LIN {X 108.19, Y 113.72, Z 0.00, A 0, B 0, C 0} C_DIS
LIN {X 108.38, Y 113.55, Z 0.00, A 0, B 0, C 0} C_DIS
LIN {X 108.56, Y 113.38, Z 0.00, A 0, B 0, C 0} C_DIS
LIN {X 108.74, Y 113.19, Z 0.00, A 0, B 0, C 0} C_DIS
LIN {X 108.92, Y 113.00, Z 0.00, A 0, B 0, C 0} C_DIS
LIN {X 109.10, Y 112.81, Z 0.00, A 0, B 0, C 0} C_DIS
LIN {X 109.28, Y 112.63, Z 0.00, A 0, B 0, C 0} C_DIS
LIN {X 109.46, Y 112.45, Z 0.00, A 0, B 0, C 0} C_DIS
LIN {X 109.65, Y 112.29, Z 0.00, A 0, B 0, C 0} C_DIS
LIN {X 109.84, Y 112.14, Z 0.00, A 0, B 0, C 0} C_DIS
LIN {X 110.04, Y 112.00, Z 0.00, A 0, B 0, C 0} C_DIS
LIN {X 110.23, Y 111.86, Z 0.00, A 0, B 0, C 0} C_DIS
LIN {X 110.42, Y 111.71, Z 0.00, A 0, B 0, C 0} C_DIS
LIN {X 110.61, Y 111.54, Z 0.00, A 0, B 0, C 0} C_DIS
LIN {X 110.79, Y 111.36, Z 0.00, A 0, B 0, C 0} C_DIS
LIN {X 110.97, Y 111.17, Z 0.00, A 0, B 0, C 0} C_DIS
LIN {X 111.15, Y 110.98, Z 0.00, A 0, B 0, C 0} C_DIS
LIN {X 111.33, Y 110.79, Z 0.00, A 0, B 0, C 0} C_DIS
LIN {X 111.51, Y 110.61, Z 0.00, A 0, B 0, C 0} C_DIS
LIN {X 111.69, Y 110.43, Z 0.00, A 0, B 0, C 0} C_DIS
LIN {X 111.88, Y 110.27, Z 0.00, A 0, B 0, C 0} C_DIS
LIN {X 112.07, Y 110.13, Z 0.00, A 0, B 0, C 0} C_DIS
LIN {X 112.27, Y 110.00, Z 0.00, A 0, B 0, C 0} C_DIS
LIN {X 112.47, Y 109.86, Z 0.00, A 0, B 0, C 0} C_DIS
LIN {X 112.65, Y 109.69, Z 0.00, A 0, B 0, C 0} C_DIS
LIN {X 112.85, Y 109.53, Z 0.00, A 0, B 0, C 0} C_DIS
LIN {X 113.05, Y 109.41, Z 0.00, A 0, B 0, C 0} C_DIS
LIN {X 113.25, Y 109.28, Z 0.00, A 0, B 0, C 0} C_DIS
LIN {X 113.42, Y 109.10, Z 0.00, A 0, B 0, C 0} C_DIS
LIN {X 113.58, Y 108.88, Z 0.00, A 0, B 0, C 0} C_DIS
LIN {X 113.74, Y 108.65, Z 0.00, A 0, B 0, C 0} C_DIS
LIN {X 113.89, Y 108.41, Z 0.00, A 0, B 0, C 0} C_DIS
LIN {X 114.02, Y 108.15, Z 0.00, A 0, B 0, C 0} C_DIS
LIN {X 114.12, Y 107.87, Z 0.00, A 0, B 0, C 0} C_DIS
LIN {X 114.20, Y 107.57, Z 0.00, A 0, B 0, C 0} C_DIS
LIN {X 114.26, Y 107.25, Z 0.00, A 0, B 0, C 0} C_DIS
LIN {X 114.30, Y 106.92, Z 0.00, A 0, B 0, C 0} C_DIS
LIN {X 114.33, Y 106.60, Z 0.00, A 0, B 0, C 0} C_DIS
LIN {X 114.36, Y 106.27, Z 0.00, A 0, B 0, C 0} C_DIS
LIN {X 114.38, Y 105.95, Z 0.00, A 0, B 0, C 0} C_DIS
LIN {X 114.39, Y 105.62, Z 0.00, A 0, B 0, C 0} C_DIS
LIN {X 114.39, Y 105.30, Z 0.00, A 0, B 0, C 0} C_DIS
LIN {X 114.40, Y 104.97, Z 0.00, A 0, B 0, C 0} C_DIS
LIN {X 114.39, Y 104.64, Z 0.00, A 0, B 0, C 0} C_DIS
LIN {X 114.39, Y 104.31, Z 0.00, A 0, B 0, C 0} C_DIS
LIN {X 114.39, Y 103.99, Z 0.00, A 0, B 0, C 0} C_DIS
LIN {X 114.38, Y 103.66, Z 0.00, A 0, B 0, C 0} C_DIS
LIN {X 114.38, Y 103.33, Z 0.00, A 0, B 0, C 0} C_DIS
LIN {X 114.38, Y 103.00, Z 0.00, A 0, B 0, C 0} C_DIS
LIN {X 114.38, Y 102.67, Z 0.00, A 0, B 0, C 0} C_DIS
LIN {X 114.38, Y 102.35, Z 0.00, A 0, B 0, C 0} C_DIS
LIN {X 114.38, Y 102.02, Z 0.00, A 0, B 0, C 0} C_DIS
LIN {X 114.39, Y 101.69, Z 0.00, A 0, B 0, C 0} C_DIS
LIN {X 114.39, Y 101.36, Z 0.00, A 0, B 0, C 0} C_DIS
LIN {X 114.39, Y 101.04, Z 0.00, A 0, B 0, C 0} C_DIS
LIN {X 114.39, Y 100.71, Z 0.00, A 0, B 0, C 0} C_DIS
LIN {X 114.39, Y 100.38, Z 0.00, A 0, B 0, C 0} C_DIS
LIN {X 114.39, Y 100.05, Z 0.00, A 0, B 0, C 0} C_DIS
LIN {X 114.39, Y 99.73, Z 0.00, A 0, B 0, C 0} C_DIS
LIN {X 114.38, Y 99.40, Z 0.00, A 0, B 0, C 0} C_DIS
LIN {X 114.38, Y 99.07, Z 0.00, A 0, B 0, C 0} C_DIS
LIN {X 114.38, Y 98.74, Z 0.00, A 0, B 0, C 0} C_DIS
LIN {X 114.38, Y 98.41, Z 0.00, A 0, B 0, C 0} C_DIS
LIN {X 114.38, Y 98.08, Z 0.00, A 0, B 0, C 0} C_DIS
LIN {X 114.39, Y 97.76, Z 0.00, A 0, B 0, C 0} C_DIS
LIN {X 114.40, Y 97.43, Z 0.00, A 0, B 0, C 0} C_DIS
LIN {X 114.42, Y 97.11, Z 0.00, A 0, B 0, C 0} C_DIS
LIN {X 114.46, Y 96.79, Z 0.00, A 0, B 0, C 0} C_DIS
LIN {X 114.54, Y 96.49, Z 0.00, A 0, B 0, C 0} C_DIS
LIN {X 114.67, Y 96.21, Z 0.00, A 0, B 0, C 0} C_DIS
LIN {X 114.82, Y 95.97, Z 0.00, A 0, B 0, C 0} C_DIS
LIN {X 115.00, Y 95.78, Z 0.00, A 0, B 0, C 0} C_DIS
LIN {X 115.19, Y 95.65, Z 0.00, A 0, B 0, C 0} C_DIS
LIN {X 115.40, Y 95.57, Z 0.00, A 0, B 0, C 0} C_DIS
LIN {X 115.61, Y 95.48, Z 0.00, A 0, B 0, C 0} C_DIS
LIN {X 115.81, Y 95.35, Z 0.00, A 0, B 0, C 0} C_DIS
LIN {X 116.01, Y 95.22, Z 0.00, A 0, B 0, C 0} C_DIS
LIN {X 116.22, Y 95.12, Z 0.00, A 0, B 0, C 0} C_DIS
LIN {X 116.43, Y 95.03, Z 0.00, A 0, B 0, C 0} C_DIS
LIN {X 116.63, Y 94.92, Z 0.00, A 0, B 0, C 0} C_DIS
LIN {X 116.83, Y 94.78, Z 0.00, A 0, B 0, C 0} C_DIS
LIN {X 117.01, Y 94.61, Z 0.00, A 0, B 0, C 0} C_DIS
LIN {X 117.20, Y 94.45, Z 0.00, A 0, B 0, C 0} C_DIS
LIN {X 117.40, Y 94.32, Z 0.00, A 0, B 0, C 0} C_DIS
LIN {X 117.60, Y 94.20, Z 0.00, A 0, B 0, C 0} C_DIS
LIN {X 117.79, Y 94.04, Z 0.00, A 0, B 0, C 0} C_DIS
LIN {X 117.97, Y 93.86, Z 0.00, A 0, B 0, C 0} C_DIS
LIN {X 118.15, Y 93.67, Z 0.00, A 0, B 0, C 0} C_DIS
LIN {X 118.33, Y 93.49, Z 0.00, A 0, B 0, C 0} C_DIS
LIN {X 118.52, Y 93.31, Z 0.00, A 0, B 0, C 0} C_DIS
LIN {X 118.70, Y 93.13, Z 0.00, A 0, B 0, C 0} C_DIS
LIN {X 118.88, Y 92.95, Z 0.00, A 0, B 0, C 0} C_DIS
LIN {X 119.06, Y 92.77, Z 0.00, A 0, B 0, C 0} C_DIS
LIN {X 119.24, Y 92.59, Z 0.00, A 0, B 0, C 0} C_DIS
LIN {X 119.42, Y 92.40, Z 0.00, A 0, B 0, C 0} C_DIS
LIN {X 119.60, Y 92.22, Z 0.00, A 0, B 0, C 0} C_DIS
LIN {X 119.78, Y 92.03, Z 0.00, A 0, B 0, C 0} C_DIS
LIN {X 119.96, Y 91.85, Z 0.00, A 0, B 0, C 0} C_DIS
LIN {X 120.14, Y 91.67, Z 0.00, A 0, B 0, C 0} C_DIS
LIN {X 120.33, Y 91.50, Z 0.00, A 0, B 0, C 0} C_DIS
LIN {X 120.51, Y 91.32, Z 0.00, A 0, B 0, C 0} C_DIS
LIN {X 120.70, Y 91.14, Z 0.00, A 0, B 0, C 0} C_DIS
LIN {X 120.87, Y 90.96, Z 0.00, A 0, B 0, C 0} C_DIS
LIN {X 121.04, Y 90.76, Z 0.00, A 0, B 0, C 0} C_DIS
LIN {X 121.21, Y 90.54, Z 0.00, A 0, B 0, C 0} C_DIS
LIN {X 121.36, Y 90.32, Z 0.00, A 0, B 0, C 0} C_DIS
LIN {X 121.52, Y 90.08, Z 0.00, A 0, B 0, C 0} C_DIS
LIN {X 121.67, Y 89.85, Z 0.00, A 0, B 0, C 0} C_DIS
LIN {X 121.83, Y 89.63, Z 0.00, A 0, B 0, C 0} C_DIS
LIN {X 121.99, Y 89.41, Z 0.00, A 0, B 0, C 0} C_DIS
LIN {X 122.16, Y 89.21, Z 0.00, A 0, B 0, C 0} C_DIS
LIN {X 122.34, Y 89.02, Z 0.00, A 0, B 0, C 0} C_DIS
LIN {X 122.52, Y 88.84, Z 0.00, A 0, B 0, C 0} C_DIS
LIN {X 122.71, Y 88.67, Z 0.00, A 0, B 0, C 0} C_DIS
LIN {X 122.89, Y 88.49, Z 0.00, A 0, B 0, C 0} C_DIS
LIN {X 123.07, Y 88.31, Z 0.00, A 0, B 0, C 0} C_DIS
LIN {X 123.24, Y 88.11, Z 0.00, A 0, B 0, C 0} C_DIS
LIN {X 123.41, Y 87.90, Z 0.00, A 0, B 0, C 0} C_DIS
LIN {X 123.56, Y 87.67, Z 0.00, A 0, B 0, C 0} C_DIS
LIN {X 123.72, Y 87.44, Z 0.00, A 0, B 0, C 0} C_DIS
LIN {X 123.87, Y 87.20, Z 0.00, A 0, B 0, C 0} C_DIS
LIN {X 124.01, Y 86.95, Z 0.00, A 0, B 0, C 0} C_DIS
LIN {X 124.13, Y 86.68, Z 0.00, A 0, B 0, C 0} C_DIS
LIN {X 124.24, Y 86.40, Z 0.00, A 0, B 0, C 0} C_DIS
LIN {X 124.36, Y 86.13, Z 0.00, A 0, B 0, C 0} C_DIS
LIN {X 124.48, Y 85.85, Z 0.00, A 0, B 0, C 0} C_DIS
LIN {X 124.60, Y 85.58, Z 0.00, A 0, B 0, C 0} C_DIS
LIN {X 124.73, Y 85.32, Z 0.00, A 0, B 0, C 0} C_DIS
LIN {X 124.87, Y 85.06, Z 0.00, A 0, B 0, C 0} C_DIS
LIN {X 125.01, Y 84.82, Z 0.00, A 0, B 0, C 0} C_DIS
LIN {X 125.16, Y 84.58, Z 0.00, A 0, B 0, C 0} C_DIS
LIN {X 125.31, Y 84.35, Z 0.00, A 0, B 0, C 0} C_DIS
LIN {X 125.47, Y 84.12, Z 0.00, A 0, B 0, C 0} C_DIS
LIN {X 125.63, Y 83.90, Z 0.00, A 0, B 0, C 0} C_DIS
LIN {X 125.79, Y 83.67, Z 0.00, A 0, B 0, C 0} C_DIS
LIN {X 125.94, Y 83.44, Z 0.00, A 0, B 0, C 0} C_DIS
LIN {X 126.08, Y 83.19, Z 0.00, A 0, B 0, C 0} C_DIS
LIN {X 126.22, Y 82.93, Z 0.00, A 0, B 0, C 0} C_DIS
LIN {X 126.34, Y 82.67, Z 0.00, A 0, B 0, C 0} C_DIS
LIN {X 126.46, Y 82.39, Z 0.00, A 0, B 0, C 0} C_DIS
LIN {X 126.57, Y 82.11, Z 0.00, A 0, B 0, C 0} C_DIS
LIN {X 126.68, Y 81.83, Z 0.00, A 0, B 0, C 0} C_DIS
LIN {X 126.77, Y 81.53, Z 0.00, A 0, B 0, C 0} C_DIS
LIN {X 126.85, Y 81.23, Z 0.00, A 0, B 0, C 0} C_DIS
LIN {X 126.95, Y 80.94, Z 0.00, A 0, B 0, C 0} C_DIS
LIN {X 127.07, Y 80.66, Z 0.00, A 0, B 0, C 0} C_DIS
LIN {X 127.19, Y 80.39, Z 0.00, A 0, B 0, C 0} C_DIS
LIN {X 127.31, Y 80.12, Z 0.00, A 0, B 0, C 0} C_DIS
LIN {X 127.43, Y 79.85, Z 0.00, A 0, B 0, C 0} C_DIS
LIN {X 127.56, Y 79.58, Z 0.00, A 0, B 0, C 0} C_DIS
LIN {X 127.68, Y 79.31, Z 0.00, A 0, B 0, C 0} C_DIS
LIN {X 127.80, Y 79.03, Z 0.00, A 0, B 0, C 0} C_DIS
LIN {X 127.91, Y 78.75, Z 0.00, A 0, B 0, C 0} C_DIS
LIN {X 128.01, Y 78.46, Z 0.00, A 0, B 0, C 0} C_DIS
LIN {X 128.10, Y 78.16, Z 0.00, A 0, B 0, C 0} C_DIS
LIN {X 128.18, Y 77.86, Z 0.00, A 0, B 0, C 0} C_DIS
LIN {X 128.29, Y 77.58, Z 0.00, A 0, B 0, C 0} C_DIS
LIN {X 128.40, Y 77.30, Z 0.00, A 0, B 0, C 0} C_DIS
LIN {X 128.49, Y 77.00, Z 0.00, A 0, B 0, C 0} C_DIS
LIN {X 128.55, Y 76.69, Z 0.00, A 0, B 0, C 0} C_DIS
LIN {X 128.61, Y 76.37, Z 0.00, A 0, B 0, C 0} C_DIS
LIN {X 128.69, Y 76.06, Z 0.00, A 0, B 0, C 0} C_DIS
LIN {X 128.78, Y 75.77, Z 0.00, A 0, B 0, C 0} C_DIS
LIN {X 128.86, Y 75.46, Z 0.00, A 0, B 0, C 0} C_DIS
LIN {X 128.91, Y 75.14, Z 0.00, A 0, B 0, C 0} C_DIS
LIN {X 128.97, Y 74.83, Z 0.00, A 0, B 0, C 0} C_DIS
LIN {X 129.07, Y 74.54, Z 0.00, A 0, B 0, C 0} C_DIS
LIN {X 129.19, Y 74.26, Z 0.00, A 0, B 0, C 0} C_DIS
LIN {X 129.29, Y 73.97, Z 0.00, A 0, B 0, C 0} C_DIS
LIN {X 129.37, Y 73.67, Z 0.00, A 0, B 0, C 0} C_DIS
LIN {X 129.43, Y 73.36, Z 0.00, A 0, B 0, C 0} C_DIS
LIN {X 129.49, Y 73.04, Z 0.00, A 0, B 0, C 0} C_DIS
LIN {X 129.54, Y 72.72, Z 0.00, A 0, B 0, C 0} C_DIS
LIN {X 129.59, Y 72.40, Z 0.00, A 0, B 0, C 0} C_DIS
LIN {X 129.64, Y 72.08, Z 0.00, A 0, B 0, C 0} C_DIS
LIN {X 129.69, Y 71.76, Z 0.00, A 0, B 0, C 0} C_DIS
LIN {X 129.75, Y 71.45, Z 0.00, A 0, B 0, C 0} C_DIS
LIN {X 129.80, Y 71.13, Z 0.00, A 0, B 0, C 0} C_DIS
LIN {X 129.85, Y 70.81, Z 0.00, A 0, B 0, C 0} C_DIS
LIN {X 129.90, Y 70.49, Z 0.00, A 0, B 0, C 0} C_DIS
LIN {X 129.96, Y 70.18, Z 0.00, A 0, B 0, C 0} C_DIS
LIN {X 130.01, Y 69.86, Z 0.00, A 0, B 0, C 0} C_DIS
LIN {X 130.06, Y 69.54, Z 0.00, A 0, B 0, C 0} C_DIS
LIN {X 130.12, Y 69.22, Z 0.00, A 0, B 0, C 0} C_DIS
LIN {X 130.17, Y 68.90, Z 0.00, A 0, B 0, C 0} C_DIS
LIN {X 130.23, Y 68.59, Z 0.00, A 0, B 0, C 0} C_DIS
LIN {X 130.28, Y 68.27, Z 0.00, A 0, B 0, C 0} C_DIS
LIN {X 130.33, Y 67.95, Z 0.00, A 0, B 0, C 0} C_DIS
LIN {X 130.38, Y 67.63, Z 0.00, A 0, B 0, C 0} C_DIS
LIN {X 130.42, Y 67.31, Z 0.00, A 0, B 0, C 0} C_DIS
LIN {X 130.45, Y 66.99, Z 0.00, A 0, B 0, C 0} C_DIS
LIN {X 130.48, Y 66.66, Z 0.00, A 0, B 0, C 0} C_DIS
LIN {X 130.49, Y 66.34, Z 0.00, A 0, B 0, C 0} C_DIS
LIN {X 130.49, Y 66.01, Z 0.00, A 0, B 0, C 0} C_DIS
LIN {X 130.49, Y 65.68, Z 0.00, A 0, B 0, C 0} C_DIS
LIN {X 130.48, Y 65.35, Z 0.00, A 0, B 0, C 0} C_DIS
LIN {X 130.47, Y 65.02, Z 0.00, A 0, B 0, C 0} C_DIS
LIN {X 130.47, Y 64.69, Z 0.00, A 0, B 0, C 0} C_DIS
LIN {X 130.47, Y 64.37, Z 0.00, A 0, B 0, C 0} C_DIS
LIN {X 130.48, Y 64.04, Z 0.00, A 0, B 0, C 0} C_DIS
LIN {X 130.50, Y 63.72, Z 0.00, A 0, B 0, C 0} C_DIS
LIN {X 130.54, Y 63.39, Z 0.00, A 0, B 0, C 0} C_DIS
LIN {X 130.58, Y 63.07, Z 0.00, A 0, B 0, C 0} C_DIS
LIN {X 130.64, Y 62.76, Z 0.00, A 0, B 0, C 0} C_DIS
LIN {X 130.70, Y 62.44, Z 0.00, A 0, B 0, C 0} C_DIS
LIN {X 130.76, Y 62.12, Z 0.00, A 0, B 0, C 0} C_DIS
LIN {X 130.81, Y 61.80, Z 0.00, A 0, B 0, C 0} C_DIS
LIN {X 130.85, Y 61.48, Z 0.00, A 0, B 0, C 0} C_DIS
LIN {X 130.88, Y 61.16, Z 0.00, A 0, B 0, C 0} C_DIS
LIN {X 130.90, Y 60.84, Z 0.00, A 0, B 0, C 0} C_DIS
LIN {X 130.91, Y 60.51, Z 0.00, A 0, B 0, C 0} C_DIS
LIN {X 130.91, Y 60.18, Z 0.00, A 0, B 0, C 0} C_DIS
LIN {X 130.92, Y 59.85, Z 0.00, A 0, B 0, C 0} C_DIS
LIN {X 130.92, Y 59.53, Z 0.00, A 0, B 0, C 0} C_DIS
LIN {X 130.92, Y 59.20, Z 0.00, A 0, B 0, C 0} C_DIS
LIN {X 130.92, Y 58.87, Z 0.00, A 0, B 0, C 0} C_DIS
LIN {X 130.92, Y 58.54, Z 0.00, A 0, B 0, C 0} C_DIS
LIN {X 130.92, Y 58.22, Z 0.00, A 0, B 0, C 0} C_DIS
LIN {X 130.91, Y 57.89, Z 0.00, A 0, B 0, C 0} C_DIS
LIN {X 130.91, Y 57.56, Z 0.00, A 0, B 0, C 0} C_DIS
LIN {X 130.91, Y 57.23, Z 0.00, A 0, B 0, C 0} C_DIS
LIN {X 130.91, Y 56.90, Z 0.00, A 0, B 0, C 0} C_DIS
LIN {X 130.91, Y 56.58, Z 0.00, A 0, B 0, C 0} C_DIS
LIN {X 130.91, Y 56.25, Z 0.00, A 0, B 0, C 0} C_DIS
LIN {X 130.91, Y 55.92, Z 0.00, A 0, B 0, C 0} C_DIS
LIN {X 130.91, Y 55.59, Z 0.00, A 0, B 0, C 0} C_DIS
LIN {X 130.91, Y 55.27, Z 0.00, A 0, B 0, C 0} C_DIS
LIN {X 130.91, Y 54.94, Z 0.00, A 0, B 0, C 0} C_DIS
LIN {X 130.91, Y 54.61, Z 0.00, A 0, B 0, C 0} C_DIS
LIN {X 130.91, Y 54.28, Z 0.00, A 0, B 0, C 0} C_DIS
LIN {X 130.91, Y 53.96, Z 0.00, A 0, B 0, C 0} C_DIS
LIN {X 130.91, Y 53.63, Z 0.00, A 0, B 0, C 0} C_DIS
LIN {X 130.91, Y 53.30, Z 0.00, A 0, B 0, C 0} C_DIS
LIN {X 130.91, Y 52.97, Z 0.00, A 0, B 0, C 0} C_DIS
LIN {X 130.91, Y 52.64, Z 0.00, A 0, B 0, C 0} C_DIS
LIN {X 130.91, Y 52.32, Z 0.00, A 0, B 0, C 0} C_DIS
LIN {X 130.91, Y 51.99, Z 0.00, A 0, B 0, C 0} C_DIS
LIN {X 130.91, Y 51.66, Z 0.00, A 0, B 0, C 0} C_DIS
LIN {X 130.91, Y 51.33, Z 0.00, A 0, B 0, C 0} C_DIS
LIN {X 130.91, Y 51.01, Z 0.00, A 0, B 0, C 0} C_DIS
LIN {X 130.91, Y 50.68, Z 0.00, A 0, B 0, C 0} C_DIS
LIN {X 130.91, Y 50.35, Z 0.00, A 0, B 0, C 0} C_DIS
LIN {X 130.91, Y 50.02, Z 0.00, A 0, B 0, C 0} C_DIS
LIN {X 130.91, Y 49.69, Z 0.00, A 0, B 0, C 0} C_DIS
LIN {X 130.91, Y 49.37, Z 0.00, A 0, B 0, C 0} C_DIS
LIN {X 130.91, Y 49.04, Z 0.00, A 0, B 0, C 0} C_DIS
LIN {X 130.91, Y 48.71, Z 0.00, A 0, B 0, C 0} C_DIS
LIN {X 130.91, Y 48.38, Z 0.00, A 0, B 0, C 0} C_DIS
LIN {X 130.91, Y 48.06, Z 0.00, A 0, B 0, C 0} C_DIS
LIN {X 130.91, Y 47.73, Z 0.00, A 0, B 0, C 0} C_DIS
LIN {X 130.91, Y 47.40, Z 0.00, A 0, B 0, C 0} C_DIS
LIN {X 130.91, Y 47.07, Z 0.00, A 0, B 0, C 0} C_DIS
LIN {X 130.91, Y 46.75, Z 0.00, A 0, B 0, C 0} C_DIS
LIN {X 130.91, Y 46.42, Z 0.00, A 0, B 0, C 0} C_DIS
LIN {X 130.91, Y 46.09, Z 0.00, A 0, B 0, C 0} C_DIS
LIN {X 130.91, Y 45.76, Z 0.00, A 0, B 0, C 0} C_DIS
LIN {X 130.91, Y 45.44, Z 0.00, A 0, B 0, C 0} C_DIS
LIN {X 130.91, Y 45.11, Z 0.00, A 0, B 0, C 0} C_DIS
LIN {X 130.91, Y 44.78, Z 0.00, A 0, B 0, C 0} C_DIS
LIN {X 130.91, Y 44.45, Z 0.00, A 0, B 0, C 0} C_DIS
LIN {X 130.91, Y 44.12, Z 0.00, A 0, B 0, C 0} C_DIS
LIN {X 130.91, Y 43.80, Z 0.00, A 0, B 0, C 0} C_DIS
LIN {X 130.91, Y 43.47, Z 0.00, A 0, B 0, C 0} C_DIS
LIN {X 130.91, Y 43.14, Z 0.00, A 0, B 0, C 0} C_DIS
LIN {X 130.91, Y 42.81, Z 0.00, A 0, B 0, C 0} C_DIS
LIN {X 130.91, Y 42.49, Z 0.00, A 0, B 0, C 0} C_DIS
LIN {X 130.91, Y 42.16, Z 0.00, A 0, B 0, C 0} C_DIS
LIN {X 130.91, Y 41.83, Z 0.00, A 0, B 0, C 0} C_DIS
LIN {X 130.91, Y 41.50, Z 0.00, A 0, B 0, C 0} C_DIS
LIN {X 130.91, Y 41.18, Z 0.00, A 0, B 0, C 0} C_DIS
LIN {X 130.91, Y 40.85, Z 0.00, A 0, B 0, C 0} C_DIS
LIN {X 130.91, Y 40.52, Z 0.00, A 0, B 0, C 0} C_DIS
LIN {X 130.91, Y 40.19, Z 0.00, A 0, B 0, C 0} C_DIS
LIN {X 130.91, Y 39.86, Z 0.00, A 0, B 0, C 0} C_DIS
LIN {X 130.91, Y 39.54, Z 0.00, A 0, B 0, C 0} C_DIS
LIN {X 130.91, Y 39.21, Z 0.00, A 0, B 0, C 0} C_DIS
LIN {X 130.91, Y 38.88, Z 0.00, A 0, B 0, C 0} C_DIS
LIN {X 130.91, Y 38.55, Z 0.00, A 0, B 0, C 0} C_DIS
LIN {X 130.91, Y 38.23, Z 0.00, A 0, B 0, C 0} C_DIS
LIN {X 130.91, Y 37.90, Z 0.00, A 0, B 0, C 0} C_DIS
LIN {X 130.91, Y 37.57, Z 0.00, A 0, B 0, C 0} C_DIS
LIN {X 130.91, Y 37.24, Z 0.00, A 0, B 0, C 0} C_DIS
LIN {X 130.91, Y 36.92, Z 0.00, A 0, B 0, C 0} C_DIS
LIN {X 130.91, Y 36.59, Z 0.00, A 0, B 0, C 0} C_DIS
LIN {X 130.91, Y 36.26, Z 0.00, A 0, B 0, C 0} C_DIS
LIN {X 130.91, Y 35.93, Z 0.00, A 0, B 0, C 0} C_DIS
LIN {X 130.91, Y 35.60, Z 0.00, A 0, B 0, C 0} C_DIS
LIN {X 130.91, Y 35.28, Z 0.00, A 0, B 0, C 0} C_DIS
LIN {X 130.91, Y 34.95, Z 0.00, A 0, B 0, C 0} C_DIS
LIN {X 130.91, Y 34.62, Z 0.00, A 0, B 0, C 0} C_DIS
LIN {X 130.91, Y 34.29, Z 0.00, A 0, B 0, C 0} C_DIS
LIN {X 130.91, Y 33.97, Z 0.00, A 0, B 0, C 0} C_DIS
LIN {X 130.91, Y 33.64, Z 0.00, A 0, B 0, C 0} C_DIS
LIN {X 130.91, Y 33.31, Z 0.00, A 0, B 0, C 0} C_DIS
LIN {X 130.91, Y 32.98, Z 0.00, A 0, B 0, C 0} C_DIS
LIN {X 130.91, Y 32.66, Z 0.00, A 0, B 0, C 0} C_DIS
LIN {X 130.91, Y 32.33, Z 0.00, A 0, B 0, C 0} C_DIS
LIN {X 130.91, Y 32.00, Z 0.00, A 0, B 0, C 0} C_DIS
LIN {X 130.91, Y 31.67, Z 0.00, A 0, B 0, C 0} C_DIS
LIN {X 130.91, Y 31.34, Z 0.00, A 0, B 0, C 0} C_DIS
LIN {X 130.91, Y 31.02, Z 0.00, A 0, B 0, C 0} C_DIS
LIN {X 130.91, Y 30.69, Z 0.00, A 0, B 0, C 0} C_DIS
LIN {X 130.91, Y 30.36, Z 0.00, A 0, B 0, C 0} C_DIS
LIN {X 130.91, Y 30.03, Z 0.00, A 0, B 0, C 0} C_DIS
LIN {X 130.91, Y 29.71, Z 0.00, A 0, B 0, C 0} C_DIS
LIN {X 130.91, Y 29.38, Z 0.00, A 0, B 0, C 0} C_DIS
LIN {X 130.91, Y 29.05, Z 0.00, A 0, B 0, C 0} C_DIS
LIN {X 130.91, Y 28.72, Z 0.00, A 0, B 0, C 0} C_DIS
LIN {X 130.91, Y 28.40, Z 0.00, A 0, B 0, C 0} C_DIS
LIN {X 130.91, Y 28.07, Z 0.00, A 0, B 0, C 0} C_DIS
LIN {X 130.91, Y 27.74, Z 0.00, A 0, B 0, C 0} C_DIS
LIN {X 130.91, Y 27.41, Z 0.00, A 0, B 0, C 0} C_DIS
LIN {X 130.91, Y 27.08, Z 0.00, A 0, B 0, C 0} C_DIS
LIN {X 130.91, Y 26.76, Z 0.00, A 0, B 0, C 0} C_DIS
LIN {X 130.91, Y 26.43, Z 0.00, A 0, B 0, C 0} C_DIS
LIN {X 130.91, Y 26.10, Z 0.00, A 0, B 0, C 0} C_DIS
LIN {X 130.91, Y 25.77, Z 0.00, A 0, B 0, C 0} C_DIS
LIN {X 130.91, Y 25.45, Z 0.00, A 0, B 0, C 0} C_DIS
LIN {X 130.91, Y 25.12, Z 0.00, A 0, B 0, C 0} C_DIS
LIN {X 130.91, Y 24.79, Z 0.00, A 0, B 0, C 0} C_DIS
LIN {X 130.91, Y 24.46, Z 0.00, A 0, B 0, C 0} C_DIS
LIN {X 130.91, Y 24.14, Z 0.00, A 0, B 0, C 0} C_DIS
LIN {X 130.91, Y 23.81, Z 0.00, A 0, B 0, C 0} C_DIS
LIN {X 130.91, Y 23.48, Z 0.00, A 0, B 0, C 0} C_DIS
LIN {X 130.91, Y 23.15, Z 0.00, A 0, B 0, C 0} C_DIS
LIN {X 130.91, Y 22.82, Z 0.00, A 0, B 0, C 0} C_DIS
LIN {X 130.91, Y 22.50, Z 0.00, A 0, B 0, C 0} C_DIS
LIN {X 130.91, Y 22.17, Z 0.00, A 0, B 0, C 0} C_DIS
LIN {X 130.91, Y 21.84, Z 0.00, A 0, B 0, C 0} C_DIS
LIN {X 130.91, Y 21.51, Z 0.00, A 0, B 0, C 0} C_DIS
LIN {X 130.91, Y 21.19, Z 0.00, A 0, B 0, C 0} C_DIS
LIN {X 130.91, Y 20.86, Z 0.00, A 0, B 0, C 0} C_DIS
LIN {X 130.91, Y 20.53, Z 0.00, A 0, B 0, C 0} C_DIS
LIN {X 130.91, Y 20.20, Z 0.00, A 0, B 0, C 0} C_DIS
LIN {X 130.91, Y 19.88, Z 0.00, A 0, B 0, C 0} C_DIS
LIN {X 130.91, Y 19.55, Z 0.00, A 0, B 0, C 0} C_DIS
LIN {X 130.91, Y 19.22, Z 0.00, A 0, B 0, C 0} C_DIS
LIN {X 130.91, Y 18.89, Z 0.00, A 0, B 0, C 0} C_DIS
LIN {X 130.91, Y 18.56, Z 0.00, A 0, B 0, C 0} C_DIS
LIN {X 130.91, Y 18.24, Z 0.00, A 0, B 0, C 0} C_DIS
LIN {X 130.91, Y 17.91, Z 0.00, A 0, B 0, C 0} C_DIS
LIN {X 130.91, Y 17.58, Z 0.00, A 0, B 0, C 0} C_DIS
LIN {X 130.91, Y 17.25, Z 0.00, A 0, B 0, C 0} C_DIS
LIN {X 130.91, Y 16.93, Z 0.00, A 0, B 0, C 0} C_DIS
LIN {X 130.91, Y 16.60, Z 0.00, A 0, B 0, C 0} C_DIS
LIN {X 130.91, Y 16.27, Z 0.00, A 0, B 0, C 0} C_DIS
LIN {X 130.91, Y 15.94, Z 0.00, A 0, B 0, C 0} C_DIS
LIN {X 130.91, Y 15.62, Z 0.00, A 0, B 0, C 0} C_DIS
LIN {X 130.91, Y 15.29, Z 0.00, A 0, B 0, C 0} C_DIS
LIN {X 130.91, Y 14.96, Z 0.00, A 0, B 0, C 0} C_DIS
LIN {X 130.91, Y 14.63, Z 0.00, A 0, B 0, C 0} C_DIS
LIN {X 130.91, Y 14.30, Z 0.00, A 0, B 0, C 0} C_DIS
LIN {X 130.91, Y 13.98, Z 0.00, A 0, B 0, C 0} C_DIS
LIN {X 130.91, Y 13.65, Z 0.00, A 0, B 0, C 0} C_DIS
LIN {X 130.91, Y 13.32, Z 0.00, A 0, B 0, C 0} C_DIS
LIN {X 130.91, Y 12.99, Z 0.00, A 0, B 0, C 0} C_DIS
LIN {X 130.91, Y 12.67, Z 0.00, A 0, B 0, C 0} C_DIS
LIN {X 130.91, Y 12.34, Z 0.00, A 0, B 0, C 0} C_DIS
LIN {X 130.91, Y 12.01, Z 0.00, A 0, B 0, C 0} C_DIS
LIN {X 130.91, Y 11.68, Z 0.00, A 0, B 0, C 0} C_DIS
LIN {X 130.91, Y 11.36, Z 0.00, A 0, B 0, C 0} C_DIS
LIN {X 130.91, Y 11.03, Z 0.00, A 0, B 0, C 0} C_DIS
LIN {X 130.91, Y 10.70, Z 0.00, A 0, B 0, C 0} C_DIS
LIN {X 130.91, Y 10.37, Z 0.00, A 0, B 0, C 0} C_DIS
LIN {X 130.91, Y 10.05, Z 0.00, A 0, B 0, C 0} C_DIS
LIN {X 130.91, Y 9.72, Z 0.00, A 0, B 0, C 0} C_DIS
LIN {X 130.91, Y 9.39, Z 0.00, A 0, B 0, C 0} C_DIS
LIN {X 130.91, Y 9.06, Z 0.00, A 0, B 0, C 0} C_DIS
LIN {X 130.91, Y 8.73, Z 0.00, A 0, B 0, C 0} C_DIS
LIN {X 130.91, Y 8.41, Z 0.00, A 0, B 0, C 0} C_DIS
LIN {X 130.91, Y 8.08, Z 0.00, A 0, B 0, C 0} C_DIS
LIN {X 130.91, Y 7.75, Z 0.00, A 0, B 0, C 0} C_DIS
LIN {X 130.91, Y 7.42, Z 0.00, A 0, B 0, C 0} C_DIS
LIN {X 130.91, Y 7.10, Z 0.00, A 0, B 0, C 0} C_DIS
LIN {X 130.91, Y 6.77, Z 0.00, A 0, B 0, C 0} C_DIS
LIN {X 130.91, Y 6.44, Z 0.00, A 0, B 0, C 0} C_DIS
LIN {X 130.91, Y 6.11, Z 0.00, A 0, B 0, C 0} C_DIS
LIN {X 130.91, Y 5.78, Z 0.00, A 0, B 0, C 0} C_DIS
LIN {X 130.91, Y 5.46, Z 0.00, A 0, B 0, C 0} C_DIS
LIN {X 130.91, Y 5.13, Z 0.00, A 0, B 0, C 0} C_DIS
LIN {X 130.91, Y 4.80, Z 0.00, A 0, B 0, C 0} C_DIS
LIN {X 130.91, Y 4.47, Z 0.00, A 0, B 0, C 0} C_DIS
LIN {X 130.91, Y 4.15, Z 0.00, A 0, B 0, C 0} C_DIS
LIN {X 130.92, Y 3.82, Z 0.00, A 0, B 0, C 0} C_DIS
LIN {X 130.92, Y 3.49, Z 0.00, A 0, B 0, C 0} C_DIS
LIN {X 130.91, Y 3.16, Z 0.00, A 0, B 0, C 0} C_DIS
LIN {X 130.91, Y 2.84, Z 0.00, A 0, B 0, C 0} C_DIS
LIN {X 130.90, Y 2.51, Z 0.00, A 0, B 0, C 0} C_DIS
LIN {X 130.88, Y 2.19, Z 0.00, A 0, B 0, C 0} C_DIS
LIN {X 130.85, Y 1.86, Z 0.00, A 0, B 0, C 0} C_DIS
LIN {X 130.81, Y 1.54, Z 0.00, A 0, B 0, C 0} C_DIS
LIN {X 130.76, Y 1.22, Z 0.00, A 0, B 0, C 0} C_DIS
LIN {X 130.71, Y 0.89, Z 0.00, A 0, B 0, C 0} C_DIS
LIN {X 130.70, Y 0.57, Z 0.00, A 0, B 0, C 0} C_DIS
LIN {X 130.76, Y 0.25, Z 0.00, A 0, B 0, C 0} C_DIS
LIN {X 130.91, Y 0.04, Z 0.00, A 0, B 0, C 0} C_DIS
LIN {X 131.12, Y -0.02, Z 0.00, A 0, B 0, C 0} C_DIS
LIN {X 131.35, Y -0.00, Z 0.00, A 0, B 0, C 0} C_DIS
LIN {X 131.56, Y 0.06, Z 0.00, A 0, B 0, C 0} C_DIS
LIN {X 131.77, Y 0.14, Z 0.00, A 0, B 0, C 0} C_DIS
LIN {X 131.98, Y 0.22, Z 0.00, A 0, B 0, C 0} C_DIS
LIN {X 132.20, Y 0.26, Z 0.00, A 0, B 0, C 0} C_DIS
LIN {X 132.42, Y 0.27, Z 0.00, A 0, B 0, C 0} C_DIS
LIN {X 132.63, Y 0.28, Z 0.00, A 0, B 0, C 0} C_DIS
LIN {X 132.85, Y 0.29, Z 0.00, A 0, B 0, C 0} C_DIS
LIN {X 133.07, Y 0.29, Z 0.00, A 0, B 0, C 0} C_DIS
LIN {X 133.29, Y 0.30, Z 0.00, A 0, B 0, C 0} C_DIS
LIN {X 133.50, Y 0.29, Z 0.00, A 0, B 0, C 0} C_DIS
LIN {X 133.72, Y 0.29, Z 0.00, A 0, B 0, C 0} C_DIS
LIN {X 133.94, Y 0.29, Z 0.00, A 0, B 0, C 0} C_DIS
LIN {X 134.16, Y 0.29, Z 0.00, A 0, B 0, C 0} C_DIS
LIN {X 134.37, Y 0.29, Z 0.00, A 0, B 0, C 0} C_DIS
LIN {X 134.59, Y 0.29, Z 0.00, A 0, B 0, C 0} C_DIS
LIN {X 134.81, Y 0.29, Z 0.00, A 0, B 0, C 0} C_DIS
LIN {X 135.03, Y 0.29, Z 0.00, A 0, B 0, C 0} C_DIS
LIN {X 135.24, Y 0.29, Z 0.00, A 0, B 0, C 0} C_DIS
LIN {X 135.46, Y 0.29, Z 0.00, A 0, B 0, C 0} C_DIS
LIN {X 135.68, Y 0.29, Z 0.00, A 0, B 0, C 0} C_DIS
LIN {X 135.90, Y 0.29, Z 0.00, A 0, B 0, C 0} C_DIS
LIN {X 136.11, Y 0.29, Z 0.00, A 0, B 0, C 0} C_DIS
LIN {X 136.33, Y 0.29, Z 0.00, A 0, B 0, C 0} C_DIS
LIN {X 136.55, Y 0.29, Z 0.00, A 0, B 0, C 0} C_DIS
LIN {X 136.77, Y 0.29, Z 0.00, A 0, B 0, C 0} C_DIS
LIN {X 136.98, Y 0.29, Z 0.00, A 0, B 0, C 0} C_DIS
LIN {X 137.20, Y 0.29, Z 0.00, A 0, B 0, C 0} C_DIS
LIN {X 137.42, Y 0.29, Z 0.00, A 0, B 0, C 0} C_DIS
LIN {X 137.64, Y 0.29, Z 0.00, A 0, B 0, C 0} C_DIS
LIN {X 137.85, Y 0.29, Z 0.00, A 0, B 0, C 0} C_DIS
LIN {X 138.07, Y 0.29, Z 0.00, A 0, B 0, C 0} C_DIS
LIN {X 138.29, Y 0.29, Z 0.00, A 0, B 0, C 0} C_DIS
LIN {X 138.50, Y 0.29, Z 0.00, A 0, B 0, C 0} C_DIS
LIN {X 138.72, Y 0.29, Z 0.00, A 0, B 0, C 0} C_DIS
LIN {X 138.94, Y 0.29, Z 0.00, A 0, B 0, C 0} C_DIS
LIN {X 139.16, Y 0.29, Z 0.00, A 0, B 0, C 0} C_DIS
LIN {X 139.37, Y 0.29, Z 0.00, A 0, B 0, C 0} C_DIS
LIN {X 139.59, Y 0.29, Z 0.00, A 0, B 0, C 0} C_DIS
LIN {X 139.81, Y 0.29, Z 0.00, A 0, B 0, C 0} C_DIS
LIN {X 140.03, Y 0.29, Z 0.00, A 0, B 0, C 0} C_DIS
LIN {X 140.24, Y 0.29, Z 0.00, A 0, B 0, C 0} C_DIS
LIN {X 140.46, Y 0.29, Z 0.00, A 0, B 0, C 0} C_DIS
LIN {X 140.68, Y 0.29, Z 0.00, A 0, B 0, C 0} C_DIS
LIN {X 140.90, Y 0.29, Z 0.00, A 0, B 0, C 0} C_DIS
LIN {X 141.11, Y 0.29, Z 0.00, A 0, B 0, C 0} C_DIS
LIN {X 141.33, Y 0.29, Z 0.00, A 0, B 0, C 0} C_DIS
LIN {X 141.55, Y 0.29, Z 0.00, A 0, B 0, C 0} C_DIS
LIN {X 141.77, Y 0.29, Z 0.00, A 0, B 0, C 0} C_DIS
LIN {X 141.98, Y 0.29, Z 0.00, A 0, B 0, C 0} C_DIS
LIN {X 142.20, Y 0.29, Z 0.00, A 0, B 0, C 0} C_DIS
LIN {X 142.42, Y 0.29, Z 0.00, A 0, B 0, C 0} C_DIS
LIN {X 142.64, Y 0.29, Z 0.00, A 0, B 0, C 0} C_DIS
LIN {X 142.85, Y 0.29, Z 0.00, A 0, B 0, C 0} C_DIS
LIN {X 143.07, Y 0.29, Z 0.00, A 0, B 0, C 0} C_DIS
LIN {X 143.29, Y 0.29, Z 0.00, A 0, B 0, C 0} C_DIS
LIN {X 143.51, Y 0.29, Z 0.00, A 0, B 0, C 0} C_DIS
LIN {X 143.72, Y 0.29, Z 0.00, A 0, B 0, C 0} C_DIS
LIN {X 143.94, Y 0.29, Z 0.00, A 0, B 0, C 0} C_DIS
LIN {X 144.16, Y 0.29, Z 0.00, A 0, B 0, C 0} C_DIS
LIN {X 144.38, Y 0.29, Z 0.00, A 0, B 0, C 0} C_DIS
LIN {X 144.59, Y 0.29, Z 0.00, A 0, B 0, C 0} C_DIS
LIN {X 144.81, Y 0.29, Z 0.00, A 0, B 0, C 0} C_DIS
LIN {X 145.03, Y 0.29, Z 0.00, A 0, B 0, C 0} C_DIS
LIN {X 145.25, Y 0.29, Z 0.00, A 0, B 0, C 0} C_DIS
LIN {X 145.46, Y 0.29, Z 0.00, A 0, B 0, C 0} C_DIS
LIN {X 145.68, Y 0.29, Z 0.00, A 0, B 0, C 0} C_DIS
LIN {X 145.90, Y 0.29, Z 0.00, A 0, B 0, C 0} C_DIS
LIN {X 146.12, Y 0.29, Z 0.00, A 0, B 0, C 0} C_DIS
LIN {X 146.33, Y 0.29, Z 0.00, A 0, B 0, C 0} C_DIS
LIN {X 146.55, Y 0.29, Z 0.00, A 0, B 0, C 0} C_DIS
LIN {X 146.77, Y 0.29, Z 0.00, A 0, B 0, C 0} C_DIS
LIN {X 146.99, Y 0.29, Z 0.00, A 0, B 0, C 0} C_DIS
LIN {X 147.20, Y 0.29, Z 0.00, A 0, B 0, C 0} C_DIS
LIN {X 147.42, Y 0.29, Z 0.00, A 0, B 0, C 0} C_DIS
LIN {X 147.64, Y 0.29, Z 0.00, A 0, B 0, C 0} C_DIS
LIN {X 147.85, Y 0.29, Z 0.00, A 0, B 0, C 0} C_DIS
LIN {X 148.07, Y 0.29, Z 0.00, A 0, B 0, C 0} C_DIS
LIN {X 148.29, Y 0.29, Z 0.00, A 0, B 0, C 0} C_DIS
LIN {X 148.51, Y 0.29, Z 0.00, A 0, B 0, C 0} C_DIS
LIN {X 148.72, Y 0.29, Z 0.00, A 0, B 0, C 0} C_DIS
LIN {X 148.94, Y 0.29, Z 0.00, A 0, B 0, C 0} C_DIS
LIN {X 149.16, Y 0.29, Z 0.00, A 0, B 0, C 0} C_DIS
LIN {X 149.38, Y 0.29, Z 0.00, A 0, B 0, C 0} C_DIS
LIN {X 149.59, Y 0.29, Z 0.00, A 0, B 0, C 0} C_DIS
LIN {X 149.81, Y 0.29, Z 0.00, A 0, B 0, C 0} C_DIS
LIN {X 150.03, Y 0.29, Z 0.00, A 0, B 0, C 0} C_DIS
LIN {X 150.25, Y 0.29, Z 0.00, A 0, B 0, C 0} C_DIS
LIN {X 150.46, Y 0.29, Z 0.00, A 0, B 0, C 0} C_DIS
LIN {X 150.68, Y 0.29, Z 0.00, A 0, B 0, C 0} C_DIS
LIN {X 150.90, Y 0.29, Z 0.00, A 0, B 0, C 0} C_DIS
LIN {X 151.12, Y 0.29, Z 0.00, A 0, B 0, C 0} C_DIS
LIN {X 151.33, Y 0.29, Z 0.00, A 0, B 0, C 0} C_DIS
LIN {X 151.55, Y 0.29, Z 0.00, A 0, B 0, C 0} C_DIS
LIN {X 151.77, Y 0.29, Z 0.00, A 0, B 0, C 0} C_DIS
LIN {X 151.99, Y 0.29, Z 0.00, A 0, B 0, C 0} C_DIS
LIN {X 152.20, Y 0.29, Z 0.00, A 0, B 0, C 0} C_DIS
LIN {X 152.42, Y 0.29, Z 0.00, A 0, B 0, C 0} C_DIS
LIN {X 152.64, Y 0.29, Z 0.00, A 0, B 0, C 0} C_DIS
LIN {X 152.86, Y 0.29, Z 0.00, A 0, B 0, C 0} C_DIS
LIN {X 153.07, Y 0.29, Z 0.00, A 0, B 0, C 0} C_DIS
LIN {X 153.29, Y 0.29, Z 0.00, A 0, B 0, C 0} C_DIS
LIN {X 153.51, Y 0.29, Z 0.00, A 0, B 0, C 0} C_DIS
LIN {X 153.73, Y 0.29, Z 0.00, A 0, B 0, C 0} C_DIS
LIN {X 153.94, Y 0.29, Z 0.00, A 0, B 0, C 0} C_DIS
LIN {X 154.16, Y 0.29, Z 0.00, A 0, B 0, C 0} C_DIS
LIN {X 154.38, Y 0.29, Z 0.00, A 0, B 0, C 0} C_DIS
LIN {X 154.60, Y 0.28, Z 0.00, A 0, B 0, C 0} C_DIS
LIN {X 154.81, Y 0.28, Z 0.00, A 0, B 0, C 0} C_DIS
LIN {X 155.03, Y 0.28, Z 0.00, A 0, B 0, C 0} C_DIS
LIN {X 155.25, Y 0.28, Z 0.00, A 0, B 0, C 0} C_DIS
LIN {X 155.47, Y 0.29, Z 0.00, A 0, B 0, C 0} C_DIS
LIN {X 155.68, Y 0.32, Z 0.00, A 0, B 0, C 0} C_DIS
LIN {X 155.89, Y 0.37, Z 0.00, A 0, B 0, C 0} C_DIS
LIN {X 156.11, Y 0.45, Z 0.00, A 0, B 0, C 0} C_DIS
LIN {X 156.32, Y 0.53, Z 0.00, A 0, B 0, C 0} C_DIS
LIN {X 156.53, Y 0.60, Z 0.00, A 0, B 0, C 0} C_DIS
LIN {X 156.74, Y 0.68, Z 0.00, A 0, B 0, C 0} C_DIS
LIN {X 156.95, Y 0.76, Z 0.00, A 0, B 0, C 0} C_DIS
LIN {X 157.16, Y 0.85, Z 0.00, A 0, B 0, C 0} C_DIS
LIN {X 157.37, Y 0.93, Z 0.00, A 0, B 0, C 0} C_DIS
LIN {X 157.58, Y 1.01, Z 0.00, A 0, B 0, C 0} C_DIS
LIN {X 157.80, Y 1.08, Z 0.00, A 0, B 0, C 0} C_DIS
LIN {X 158.01, Y 1.15, Z 0.00, A 0, B 0, C 0} C_DIS
LIN {X 158.22, Y 1.22, Z 0.00, A 0, B 0, C 0} C_DIS
LIN {X 158.43, Y 1.32, Z 0.00, A 0, B 0, C 0} C_DIS
LIN {X 158.63, Y 1.43, Z 0.00, A 0, B 0, C 0} C_DIS
LIN {X 158.84, Y 1.54, Z 0.00, A 0, B 0, C 0} C_DIS
LIN {X 159.04, Y 1.66, Z 0.00, A 0, B 0, C 0} C_DIS
LIN {X 159.24, Y 1.77, Z 0.00, A 0, B 0, C 0} C_DIS
LIN {X 159.45, Y 1.87, Z 0.00, A 0, B 0, C 0} C_DIS
LIN {X 159.66, Y 1.97, Z 0.00, A 0, B 0, C 0} C_DIS
LIN {X 159.85, Y 2.10, Z 0.00, A 0, B 0, C 0} C_DIS
LIN {X 160.04, Y 2.27, Z 0.00, A 0, B 0, C 0} C_DIS
LIN {X 160.23, Y 2.43, Z 0.00, A 0, B 0, C 0} C_DIS
LIN {X 160.43, Y 2.56, Z 0.00, A 0, B 0, C 0} C_DIS
LIN {X 160.63, Y 2.69, Z 0.00, A 0, B 0, C 0} C_DIS
LIN {X 160.82, Y 2.84, Z 0.00, A 0, B 0, C 0} C_DIS
LIN {X 161.00, Y 3.02, Z 0.00, A 0, B 0, C 0} C_DIS
LIN {X 161.18, Y 3.20, Z 0.00, A 0, B 0, C 0} C_DIS
LIN {X 161.36, Y 3.39, Z 0.00, A 0, B 0, C 0} C_DIS
LIN {X 161.54, Y 3.57, Z 0.00, A 0, B 0, C 0} C_DIS
LIN {X 161.72, Y 3.75, Z 0.00, A 0, B 0, C 0} C_DIS
LIN {X 161.90, Y 3.93, Z 0.00, A 0, B 0, C 0} C_DIS
LIN {X 162.08, Y 4.11, Z 0.00, A 0, B 0, C 0} C_DIS
LIN {X 162.27, Y 4.29, Z 0.00, A 0, B 0, C 0} C_DIS
LIN {X 162.45, Y 4.47, Z 0.00, A 0, B 0, C 0} C_DIS
LIN {X 162.63, Y 4.65, Z 0.00, A 0, B 0, C 0} C_DIS
LIN {X 162.80, Y 4.85, Z 0.00, A 0, B 0, C 0} C_DIS
LIN {X 162.96, Y 5.07, Z 0.00, A 0, B 0, C 0} C_DIS
LIN {X 163.12, Y 5.30, Z 0.00, A 0, B 0, C 0} C_DIS
LIN {X 163.28, Y 5.52, Z 0.00, A 0, B 0, C 0} C_DIS
LIN {X 163.45, Y 5.72, Z 0.00, A 0, B 0, C 0} C_DIS
LIN {X 163.63, Y 5.90, Z 0.00, A 0, B 0, C 0} C_DIS
LIN {X 163.81, Y 6.08, Z 0.00, A 0, B 0, C 0} C_DIS
LIN {X 164.00, Y 6.25, Z 0.00, A 0, B 0, C 0} C_DIS
LIN {X 164.18, Y 6.43, Z 0.00, A 0, B 0, C 0} C_DIS
LIN {X 164.36, Y 6.61, Z 0.00, A 0, B 0, C 0} C_DIS
LIN {X 164.54, Y 6.81, Z 0.00, A 0, B 0, C 0} C_DIS
LIN {X 164.70, Y 7.02, Z 0.00, A 0, B 0, C 0} C_DIS
LIN {X 164.85, Y 7.25, Z 0.00, A 0, B 0, C 0} C_DIS
LIN {X 165.01, Y 7.49, Z 0.00, A 0, B 0, C 0} C_DIS
LIN {X 165.16, Y 7.72, Z 0.00, A 0, B 0, C 0} C_DIS
LIN {X 165.31, Y 7.95, Z 0.00, A 0, B 0, C 0} C_DIS
LIN {X 165.47, Y 8.19, Z 0.00, A 0, B 0, C 0} C_DIS
LIN {X 165.62, Y 8.42, Z 0.00, A 0, B 0, C 0} C_DIS
LIN {X 165.77, Y 8.65, Z 0.00, A 0, B 0, C 0} C_DIS
LIN {X 165.93, Y 8.88, Z 0.00, A 0, B 0, C 0} C_DIS
LIN {X 166.08, Y 9.11, Z 0.00, A 0, B 0, C 0} C_DIS
LIN {X 166.24, Y 9.34, Z 0.00, A 0, B 0, C 0} C_DIS
LIN {X 166.39, Y 9.57, Z 0.00, A 0, B 0, C 0} C_DIS
LIN {X 166.54, Y 9.81, Z 0.00, A 0, B 0, C 0} C_DIS
LIN {X 166.70, Y 10.04, Z 0.00, A 0, B 0, C 0} C_DIS
LIN {X 166.85, Y 10.27, Z 0.00, A 0, B 0, C 0} C_DIS
LIN {X 167.00, Y 10.50, Z 0.00, A 0, B 0, C 0} C_DIS
LIN {X 167.16, Y 10.73, Z 0.00, A 0, B 0, C 0} C_DIS
LIN {X 167.31, Y 10.96, Z 0.00, A 0, B 0, C 0} C_DIS
LIN {X 167.47, Y 11.20, Z 0.00, A 0, B 0, C 0} C_DIS
LIN {X 167.62, Y 11.43, Z 0.00, A 0, B 0, C 0} C_DIS
LIN {X 167.77, Y 11.66, Z 0.00, A 0, B 0, C 0} C_DIS
LIN {X 167.93, Y 11.89, Z 0.00, A 0, B 0, C 0} C_DIS
LIN {X 168.08, Y 12.12, Z 0.00, A 0, B 0, C 0} C_DIS
LIN {X 168.23, Y 12.36, Z 0.00, A 0, B 0, C 0} C_DIS
LIN {X 168.39, Y 12.59, Z 0.00, A 0, B 0, C 0} C_DIS
LIN {X 168.54, Y 12.82, Z 0.00, A 0, B 0, C 0} C_DIS
LIN {X 168.70, Y 13.05, Z 0.00, A 0, B 0, C 0} C_DIS
LIN {X 168.85, Y 13.28, Z 0.00, A 0, B 0, C 0} C_DIS
LIN {X 169.00, Y 13.51, Z 0.00, A 0, B 0, C 0} C_DIS
LIN {X 169.16, Y 13.75, Z 0.00, A 0, B 0, C 0} C_DIS
LIN {X 169.31, Y 13.98, Z 0.00, A 0, B 0, C 0} C_DIS
LIN {X 169.46, Y 14.21, Z 0.00, A 0, B 0, C 0} C_DIS
LIN {X 169.62, Y 14.44, Z 0.00, A 0, B 0, C 0} C_DIS
LIN {X 169.77, Y 14.67, Z 0.00, A 0, B 0, C 0} C_DIS
LIN {X 169.93, Y 14.90, Z 0.00, A 0, B 0, C 0} C_DIS
LIN {X 170.08, Y 15.14, Z 0.00, A 0, B 0, C 0} C_DIS
LIN {X 170.23, Y 15.37, Z 0.00, A 0, B 0, C 0} C_DIS
LIN {X 170.39, Y 15.60, Z 0.00, A 0, B 0, C 0} C_DIS
LIN {X 170.54, Y 15.83, Z 0.00, A 0, B 0, C 0} C_DIS
LIN {X 170.69, Y 16.06, Z 0.00, A 0, B 0, C 0} C_DIS
LIN {X 170.85, Y 16.29, Z 0.00, A 0, B 0, C 0} C_DIS
LIN {X 171.00, Y 16.53, Z 0.00, A 0, B 0, C 0} C_DIS
LIN {X 171.16, Y 16.76, Z 0.00, A 0, B 0, C 0} C_DIS
LIN {X 171.31, Y 16.99, Z 0.00, A 0, B 0, C 0} C_DIS
LIN {X 171.46, Y 17.22, Z 0.00, A 0, B 0, C 0} C_DIS
LIN {X 171.62, Y 17.45, Z 0.00, A 0, B 0, C 0} C_DIS
LIN {X 171.77, Y 17.68, Z 0.00, A 0, B 0, C 0} C_DIS
LIN {X 171.92, Y 17.92, Z 0.00, A 0, B 0, C 0} C_DIS
LIN {X 172.08, Y 18.15, Z 0.00, A 0, B 0, C 0} C_DIS
LIN {X 172.23, Y 18.38, Z 0.00, A 0, B 0, C 0} C_DIS
LIN {X 172.39, Y 18.61, Z 0.00, A 0, B 0, C 0} C_DIS
LIN {X 172.54, Y 18.84, Z 0.00, A 0, B 0, C 0} C_DIS
LIN {X 172.69, Y 19.07, Z 0.00, A 0, B 0, C 0} C_DIS
LIN {X 172.85, Y 19.31, Z 0.00, A 0, B 0, C 0} C_DIS
LIN {X 173.00, Y 19.54, Z 0.00, A 0, B 0, C 0} C_DIS
LIN {X 173.15, Y 19.77, Z 0.00, A 0, B 0, C 0} C_DIS
LIN {X 173.31, Y 20.00, Z 0.00, A 0, B 0, C 0} C_DIS
LIN {X 173.46, Y 20.23, Z 0.00, A 0, B 0, C 0} C_DIS
LIN {X 173.62, Y 20.47, Z 0.00, A 0, B 0, C 0} C_DIS
LIN {X 173.77, Y 20.70, Z 0.00, A 0, B 0, C 0} C_DIS
LIN {X 173.92, Y 20.93, Z 0.00, A 0, B 0, C 0} C_DIS
LIN {X 174.08, Y 21.16, Z 0.00, A 0, B 0, C 0} C_DIS
LIN {X 174.23, Y 21.39, Z 0.00, A 0, B 0, C 0} C_DIS
LIN {X 174.38, Y 21.62, Z 0.00, A 0, B 0, C 0} C_DIS
LIN {X 174.54, Y 21.86, Z 0.00, A 0, B 0, C 0} C_DIS
LIN {X 174.69, Y 22.09, Z 0.00, A 0, B 0, C 0} C_DIS
LIN {X 174.85, Y 22.32, Z 0.00, A 0, B 0, C 0} C_DIS
LIN {X 175.00, Y 22.55, Z 0.00, A 0, B 0, C 0} C_DIS
LIN {X 175.15, Y 22.78, Z 0.00, A 0, B 0, C 0} C_DIS
LIN {X 175.31, Y 23.01, Z 0.00, A 0, B 0, C 0} C_DIS
LIN {X 175.46, Y 23.24, Z 0.00, A 0, B 0, C 0} C_DIS
LIN {X 175.61, Y 23.48, Z 0.00, A 0, B 0, C 0} C_DIS
LIN {X 175.77, Y 23.71, Z 0.00, A 0, B 0, C 0} C_DIS
LIN {X 175.92, Y 23.94, Z 0.00, A 0, B 0, C 0} C_DIS
LIN {X 176.07, Y 24.17, Z 0.00, A 0, B 0, C 0} C_DIS
LIN {X 176.23, Y 24.41, Z 0.00, A 0, B 0, C 0} C_DIS
LIN {X 176.38, Y 24.64, Z 0.00, A 0, B 0, C 0} C_DIS
LIN {X 176.54, Y 24.87, Z 0.00, A 0, B 0, C 0} C_DIS
LIN {X 176.70, Y 25.09, Z 0.00, A 0, B 0, C 0} C_DIS
LIN {X 176.86, Y 25.30, Z 0.00, A 0, B 0, C 0} C_DIS
LIN {X 177.04, Y 25.49, Z 0.00, A 0, B 0, C 0} C_DIS
LIN {X 177.22, Y 25.67, Z 0.00, A 0, B 0, C 0} C_DIS
LIN {X 177.40, Y 25.84, Z 0.00, A 0, B 0, C 0} C_DIS
LIN {X 177.59, Y 26.02, Z 0.00, A 0, B 0, C 0} C_DIS
LIN {X 177.77, Y 26.19, Z 0.00, A 0, B 0, C 0} C_DIS
LIN {X 177.95, Y 26.39, Z 0.00, A 0, B 0, C 0} C_DIS
LIN {X 178.11, Y 26.60, Z 0.00, A 0, B 0, C 0} C_DIS
LIN {X 178.27, Y 26.82, Z 0.00, A 0, B 0, C 0} C_DIS
LIN {X 178.43, Y 27.05, Z 0.00, A 0, B 0, C 0} C_DIS
LIN {X 178.59, Y 27.26, Z 0.00, A 0, B 0, C 0} C_DIS
LIN {X 178.77, Y 27.45, Z 0.00, A 0, B 0, C 0} C_DIS
LIN {X 178.95, Y 27.63, Z 0.00, A 0, B 0, C 0} C_DIS
LIN {X 179.14, Y 27.80, Z 0.00, A 0, B 0, C 0} C_DIS
LIN {X 179.32, Y 27.98, Z 0.00, A 0, B 0, C 0} C_DIS
LIN {X 179.50, Y 28.16, Z 0.00, A 0, B 0, C 0} C_DIS
LIN {X 179.68, Y 28.34, Z 0.00, A 0, B 0, C 0} C_DIS
LIN {X 179.86, Y 28.52, Z 0.00, A 0, B 0, C 0} C_DIS
LIN {X 180.04, Y 28.71, Z 0.00, A 0, B 0, C 0} C_DIS
LIN {X 180.22, Y 28.89, Z 0.00, A 0, B 0, C 0} C_DIS
LIN {X 180.41, Y 29.07, Z 0.00, A 0, B 0, C 0} C_DIS
LIN {X 180.59, Y 29.25, Z 0.00, A 0, B 0, C 0} C_DIS
LIN {X 180.77, Y 29.44, Z 0.00, A 0, B 0, C 0} C_DIS
LIN {X 180.95, Y 29.62, Z 0.00, A 0, B 0, C 0} C_DIS
LIN {X 181.13, Y 29.80, Z 0.00, A 0, B 0, C 0} C_DIS
LIN {X 181.31, Y 29.99, Z 0.00, A 0, B 0, C 0} C_DIS
LIN {X 181.49, Y 30.17, Z 0.00, A 0, B 0, C 0} C_DIS
LIN {X 181.67, Y 30.35, Z 0.00, A 0, B 0, C 0} C_DIS
LIN {X 181.86, Y 30.51, Z 0.00, A 0, B 0, C 0} C_DIS
LIN {X 182.05, Y 30.67, Z 0.00, A 0, B 0, C 0} C_DIS
LIN {X 182.25, Y 30.80, Z 0.00, A 0, B 0, C 0} C_DIS
LIN {X 182.45, Y 30.93, Z 0.00, A 0, B 0, C 0} C_DIS
LIN {X 182.63, Y 31.09, Z 0.00, A 0, B 0, C 0} C_DIS
LIN {X 182.82, Y 31.25, Z 0.00, A 0, B 0, C 0} C_DIS
LIN {X 183.02, Y 31.39, Z 0.00, A 0, B 0, C 0} C_DIS
LIN {X 183.22, Y 31.51, Z 0.00, A 0, B 0, C 0} C_DIS
LIN {X 183.41, Y 31.67, Z 0.00, A 0, B 0, C 0} C_DIS
LIN {X 183.60, Y 31.83, Z 0.00, A 0, B 0, C 0} C_DIS
LIN {X 183.79, Y 31.98, Z 0.00, A 0, B 0, C 0} C_DIS
LIN {X 183.99, Y 32.11, Z 0.00, A 0, B 0, C 0} C_DIS
LIN {X 184.19, Y 32.24, Z 0.00, A 0, B 0, C 0} C_DIS
LIN {X 184.38, Y 32.41, Z 0.00, A 0, B 0, C 0} C_DIS
LIN {X 184.57, Y 32.57, Z 0.00, A 0, B 0, C 0} C_DIS
LIN {X 184.77, Y 32.70, Z 0.00, A 0, B 0, C 0} C_DIS
LIN {X 184.97, Y 32.79, Z 0.00, A 0, B 0, C 0} C_DIS
LIN {X 185.18, Y 32.89, Z 0.00, A 0, B 0, C 0} C_DIS
LIN {X 185.38, Y 33.00, Z 0.00, A 0, B 0, C 0} C_DIS
LIN {X 185.58, Y 33.13, Z 0.00, A 0, B 0, C 0} C_DIS
LIN {X 185.78, Y 33.25, Z 0.00, A 0, B 0, C 0} C_DIS
LIN {X 186.00, Y 33.33, Z 0.00, A 0, B 0, C 0} C_DIS
LIN {X 186.20, Y 33.43, Z 0.00, A 0, B 0, C 0} C_DIS
LIN {X 186.39, Y 33.58, Z 0.00, A 0, B 0, C 0} C_DIS
LIN {X 186.58, Y 33.75, Z 0.00, A 0, B 0, C 0} C_DIS
LIN {X 186.77, Y 33.90, Z 0.00, A 0, B 0, C 0} C_DIS
LIN {X 186.97, Y 34.02, Z 0.00, A 0, B 0, C 0} C_DIS
LIN {X 187.18, Y 34.12, Z 0.00, A 0, B 0, C 0} C_DIS
LIN {X 187.39, Y 34.20, Z 0.00, A 0, B 0, C 0} C_DIS
LIN {X 187.60, Y 34.28, Z 0.00, A 0, B 0, C 0} C_DIS
LIN {X 187.82, Y 34.35, Z 0.00, A 0, B 0, C 0} C_DIS
LIN {X 188.03, Y 34.43, Z 0.00, A 0, B 0, C 0} C_DIS
LIN {X 188.24, Y 34.51, Z 0.00, A 0, B 0, C 0} C_DIS
LIN {X 188.45, Y 34.59, Z 0.00, A 0, B 0, C 0} C_DIS
LIN {X 188.66, Y 34.67, Z 0.00, A 0, B 0, C 0} C_DIS
LIN {X 188.87, Y 34.74, Z 0.00, A 0, B 0, C 0} C_DIS
LIN {X 189.08, Y 34.84, Z 0.00, A 0, B 0, C 0} C_DIS
LIN {X 189.28, Y 34.96, Z 0.00, A 0, B 0, C 0} C_DIS
LIN {X 189.48, Y 35.09, Z 0.00, A 0, B 0, C 0} C_DIS
LIN {X 189.68, Y 35.20, Z 0.00, A 0, B 0, C 0} C_DIS
LIN {X 189.89, Y 35.30, Z 0.00, A 0, B 0, C 0} C_DIS
LIN {X 190.10, Y 35.39, Z 0.00, A 0, B 0, C 0} C_DIS
LIN {X 190.31, Y 35.47, Z 0.00, A 0, B 0, C 0} C_DIS
LIN {X 190.52, Y 35.54, Z 0.00, A 0, B 0, C 0} C_DIS
LIN {X 190.74, Y 35.59, Z 0.00, A 0, B 0, C 0} C_DIS
LIN {X 190.95, Y 35.65, Z 0.00, A 0, B 0, C 0} C_DIS
LIN {X 191.17, Y 35.69, Z 0.00, A 0, B 0, C 0} C_DIS
LIN {X 191.38, Y 35.74, Z 0.00, A 0, B 0, C 0} C_DIS
LIN {X 191.60, Y 35.78, Z 0.00, A 0, B 0, C 0} C_DIS
LIN {X 191.81, Y 35.84, Z 0.00, A 0, B 0, C 0} C_DIS
LIN {X 192.02, Y 35.92, Z 0.00, A 0, B 0, C 0} C_DIS
LIN {X 192.23, Y 36.01, Z 0.00, A 0, B 0, C 0} C_DIS
LIN {X 192.44, Y 36.10, Z 0.00, A 0, B 0, C 0} C_DIS
LIN {X 192.65, Y 36.18, Z 0.00, A 0, B 0, C 0} C_DIS
LIN {X 192.86, Y 36.25, Z 0.00, A 0, B 0, C 0} C_DIS
LIN {X 193.08, Y 36.30, Z 0.00, A 0, B 0, C 0} C_DIS
LIN {X 193.29, Y 36.33, Z 0.00, A 0, B 0, C 0} C_DIS
LIN {X 193.51, Y 36.35, Z 0.00, A 0, B 0, C 0} C_DIS
LIN {X 193.73, Y 36.35, Z 0.00, A 0, B 0, C 0} C_DIS
LIN {X 193.95, Y 36.34, Z 0.00, A 0, B 0, C 0} C_DIS
LIN {X 194.17, Y 36.33, Z 0.00, A 0, B 0, C 0} C_DIS
LIN {X 194.38, Y 36.32, Z 0.00, A 0, B 0, C 0} C_DIS
LIN {X 194.60, Y 36.33, Z 0.00, A 0, B 0, C 0} C_DIS
LIN {X 194.81, Y 36.37, Z 0.00, A 0, B 0, C 0} C_DIS
LIN {X 195.03, Y 36.43, Z 0.00, A 0, B 0, C 0} C_DIS
LIN {X 195.24, Y 36.50, Z 0.00, A 0, B 0, C 0} C_DIS
LIN {X 195.45, Y 36.56, Z 0.00, A 0, B 0, C 0} C_DIS
LIN {X 195.67, Y 36.64, Z 0.00, A 0, B 0, C 0} C_DIS
LIN {X 195.88, Y 36.72, Z 0.00, A 0, B 0, C 0} C_DIS
LIN {X 196.08, Y 36.83, Z 0.00, A 0, B 0, C 0} C_DIS
LIN {X 196.28, Y 36.96, Z 0.00, A 0, B 0, C 0} C_DIS
LIN {X 196.47, Y 37.12, Z 0.00, A 0, B 0, C 0} C_DIS
LIN {X 196.64, Y 37.32, Z 0.00, A 0, B 0, C 0} C_DIS
LIN {X 196.79, Y 37.56, Z 0.00, A 0, B 0, C 0} C_DIS
LIN {X 196.91, Y 37.83, Z 0.00, A 0, B 0, C 0} C_DIS
LIN {X 197.01, Y 38.12, Z 0.00, A 0, B 0, C 0} C_DIS
LIN {X 197.08, Y 38.44, Z 0.00, A 0, B 0, C 0} C_DIS
LIN {X 197.13, Y 38.75, Z 0.00, A 0, B 0, C 0} C_DIS
LIN {X 197.20, Y 39.06, Z 0.00, A 0, B 0, C 0} C_DIS
LIN {X 197.30, Y 39.35, Z 0.00, A 0, B 0, C 0} C_DIS
LIN {X 197.41, Y 39.63, Z 0.00, A 0, B 0, C 0} C_DIS
LIN {X 197.51, Y 39.92, Z 0.00, A 0, B 0, C 0} C_DIS
LIN {X 197.60, Y 40.22, Z 0.00, A 0, B 0, C 0} C_DIS
LIN {X 197.69, Y 40.52, Z 0.00, A 0, B 0, C 0} C_DIS
LIN {X 197.79, Y 40.81, Z 0.00, A 0, B 0, C 0} C_DIS
LIN {X 197.90, Y 41.09, Z 0.00, A 0, B 0, C 0} C_DIS
LIN {X 198.02, Y 41.36, Z 0.00, A 0, B 0, C 0} C_DIS
LIN {X 198.15, Y 41.63, Z 0.00, A 0, B 0, C 0} C_DIS
LIN {X 198.29, Y 41.88, Z 0.00, A 0, B 0, C 0} C_DIS
LIN {X 198.43, Y 42.13, Z 0.00, A 0, B 0, C 0} C_DIS
LIN {X 198.58, Y 42.37, Z 0.00, A 0, B 0, C 0} C_DIS
LIN {X 198.73, Y 42.60, Z 0.00, A 0, B 0, C 0} C_DIS
LIN {X 198.88, Y 42.83, Z 0.00, A 0, B 0, C 0} C_DIS
LIN {X 199.04, Y 43.06, Z 0.00, A 0, B 0, C 0} C_DIS
LIN {X 199.20, Y 43.29, Z 0.00, A 0, B 0, C 0} C_DIS
LIN {X 199.35, Y 43.52, Z 0.00, A 0, B 0, C 0} C_DIS
LIN {X 199.51, Y 43.75, Z 0.00, A 0, B 0, C 0} C_DIS
LIN {X 199.66, Y 43.98, Z 0.00, A 0, B 0, C 0} C_DIS
LIN {X 199.82, Y 44.21, Z 0.00, A 0, B 0, C 0} C_DIS
LIN {X 199.97, Y 44.44, Z 0.00, A 0, B 0, C 0} C_DIS
LIN {X 200.12, Y 44.67, Z 0.00, A 0, B 0, C 0} C_DIS
LIN {X 200.27, Y 44.91, Z 0.00, A 0, B 0, C 0} C_DIS
LIN {X 200.42, Y 45.15, Z 0.00, A 0, B 0, C 0} C_DIS
LIN {X 200.57, Y 45.39, Z 0.00, A 0, B 0, C 0} C_DIS
LIN {X 200.73, Y 45.62, Z 0.00, A 0, B 0, C 0} C_DIS
LIN {X 200.89, Y 45.84, Z 0.00, A 0, B 0, C 0} C_DIS
LIN {X 201.05, Y 46.05, Z 0.00, A 0, B 0, C 0} C_DIS
LIN {X 201.22, Y 46.25, Z 0.00, A 0, B 0, C 0} C_DIS
LIN {X 201.40, Y 46.44, Z 0.00, A 0, B 0, C 0} C_DIS
LIN {X 201.57, Y 46.64, Z 0.00, A 0, B 0, C 0} C_DIS
LIN {X 201.74, Y 46.84, Z 0.00, A 0, B 0, C 0} C_DIS
LIN {X 201.87, Y 47.11, Z 0.00, A 0, B 0, C 0} C_DIS
LIN {X 201.91, Y 47.43, Z 0.00, A 0, B 0, C 0} C_DIS
LIN {X 201.86, Y 47.74, Z 0.00, A 0, B 0, C 0} C_DIS
LIN {X 201.75, Y 48.03, Z 0.00, A 0, B 0, C 0} C_DIS
LIN {X 201.62, Y 48.30, Z 0.00, A 0, B 0, C 0} C_DIS
LIN {X 201.50, Y 48.58, Z 0.00, A 0, B 0, C 0} C_DIS
LIN {X 201.38, Y 48.85, Z 0.00, A 0, B 0, C 0} C_DIS
LIN {X 201.26, Y 49.12, Z 0.00, A 0, B 0, C 0} C_DIS
LIN {X 201.14, Y 49.39, Z 0.00, A 0, B 0, C 0} C_DIS
LIN {X 201.02, Y 49.66, Z 0.00, A 0, B 0, C 0} C_DIS
LIN {X 200.90, Y 49.93, Z 0.00, A 0, B 0, C 0} C_DIS
LIN {X 200.79, Y 50.22, Z 0.00, A 0, B 0, C 0} C_DIS
LIN {X 200.69, Y 50.51, Z 0.00, A 0, B 0, C 0} C_DIS
LIN {X 200.60, Y 50.81, Z 0.00, A 0, B 0, C 0} C_DIS
LIN {X 200.51, Y 51.10, Z 0.00, A 0, B 0, C 0} C_DIS
LIN {X 200.41, Y 51.39, Z 0.00, A 0, B 0, C 0} C_DIS
LIN {X 200.29, Y 51.66, Z 0.00, A 0, B 0, C 0} C_DIS
LIN {X 200.17, Y 51.94, Z 0.00, A 0, B 0, C 0} C_DIS
LIN {X 200.05, Y 52.21, Z 0.00, A 0, B 0, C 0} C_DIS
LIN {X 199.92, Y 52.47, Z 0.00, A 0, B 0, C 0} C_DIS
LIN {X 199.79, Y 52.74, Z 0.00, A 0, B 0, C 0} C_DIS
LIN {X 199.67, Y 53.01, Z 0.00, A 0, B 0, C 0} C_DIS
LIN {X 199.56, Y 53.29, Z 0.00, A 0, B 0, C 0} C_DIS
LIN {X 199.46, Y 53.58, Z 0.00, A 0, B 0, C 0} C_DIS
LIN {X 199.36, Y 53.88, Z 0.00, A 0, B 0, C 0} C_DIS
LIN {X 199.27, Y 54.17, Z 0.00, A 0, B 0, C 0} C_DIS
LIN {X 199.17, Y 54.46, Z 0.00, A 0, B 0, C 0} C_DIS
LIN {X 199.07, Y 54.75, Z 0.00, A 0, B 0, C 0} C_DIS
LIN {X 198.95, Y 55.02, Z 0.00, A 0, B 0, C 0} C_DIS
LIN {X 198.83, Y 55.29, Z 0.00, A 0, B 0, C 0} C_DIS
LIN {X 198.70, Y 55.56, Z 0.00, A 0, B 0, C 0} C_DIS
LIN {X 198.58, Y 55.83, Z 0.00, A 0, B 0, C 0} C_DIS
LIN {X 198.45, Y 56.10, Z 0.00, A 0, B 0, C 0} C_DIS
LIN {X 198.33, Y 56.38, Z 0.00, A 0, B 0, C 0} C_DIS
LIN {X 198.22, Y 56.66, Z 0.00, A 0, B 0, C 0} C_DIS
LIN {X 198.12, Y 56.94, Z 0.00, A 0, B 0, C 0} C_DIS
LIN {X 198.03, Y 57.24, Z 0.00, A 0, B 0, C 0} C_DIS
LIN {X 197.94, Y 57.54, Z 0.00, A 0, B 0, C 0} C_DIS
LIN {X 197.85, Y 57.83, Z 0.00, A 0, B 0, C 0} C_DIS
LIN {X 197.73, Y 58.11, Z 0.00, A 0, B 0, C 0} C_DIS
LIN {X 197.60, Y 58.38, Z 0.00, A 0, B 0, C 0} C_DIS
LIN {X 197.48, Y 58.65, Z 0.00, A 0, B 0, C 0} C_DIS
LIN {X 197.36, Y 58.92, Z 0.00, A 0, B 0, C 0} C_DIS
LIN {X 197.24, Y 59.19, Z 0.00, A 0, B 0, C 0} C_DIS
LIN {X 197.12, Y 59.46, Z 0.00, A 0, B 0, C 0} C_DIS
LIN {X 197.00, Y 59.74, Z 0.00, A 0, B 0, C 0} C_DIS
LIN {X 196.88, Y 60.02, Z 0.00, A 0, B 0, C 0} C_DIS
LIN {X 196.76, Y 60.29, Z 0.00, A 0, B 0, C 0} C_DIS
LIN {X 196.64, Y 60.56, Z 0.00, A 0, B 0, C 0} C_DIS
LIN {X 196.51, Y 60.82, Z 0.00, A 0, B 0, C 0} C_DIS
LIN {X 196.36, Y 61.06, Z 0.00, A 0, B 0, C 0} C_DIS
LIN {X 196.21, Y 61.29, Z 0.00, A 0, B 0, C 0} C_DIS
LIN {X 196.06, Y 61.52, Z 0.00, A 0, B 0, C 0} C_DIS
LIN {X 195.90, Y 61.75, Z 0.00, A 0, B 0, C 0} C_DIS
LIN {X 195.75, Y 61.99, Z 0.00, A 0, B 0, C 0} C_DIS
LIN {X 195.59, Y 62.22, Z 0.00, A 0, B 0, C 0} C_DIS
LIN {X 195.44, Y 62.45, Z 0.00, A 0, B 0, C 0} C_DIS
LIN {X 195.29, Y 62.68, Z 0.00, A 0, B 0, C 0} C_DIS
LIN {X 195.13, Y 62.92, Z 0.00, A 0, B 0, C 0} C_DIS
LIN {X 194.98, Y 63.15, Z 0.00, A 0, B 0, C 0} C_DIS
LIN {X 194.83, Y 63.38, Z 0.00, A 0, B 0, C 0} C_DIS
LIN {X 194.67, Y 63.61, Z 0.00, A 0, B 0, C 0} C_DIS
LIN {X 194.52, Y 63.84, Z 0.00, A 0, B 0, C 0} C_DIS
LIN {X 194.36, Y 64.07, Z 0.00, A 0, B 0, C 0} C_DIS
LIN {X 194.21, Y 64.30, Z 0.00, A 0, B 0, C 0} C_DIS
LIN {X 194.05, Y 64.53, Z 0.00, A 0, B 0, C 0} C_DIS
LIN {X 193.90, Y 64.77, Z 0.00, A 0, B 0, C 0} C_DIS
LIN {X 193.75, Y 65.00, Z 0.00, A 0, B 0, C 0} C_DIS
LIN {X 193.59, Y 65.23, Z 0.00, A 0, B 0, C 0} C_DIS
LIN {X 193.44, Y 65.46, Z 0.00, A 0, B 0, C 0} C_DIS
LIN {X 193.29, Y 65.70, Z 0.00, A 0, B 0, C 0} C_DIS
LIN {X 193.14, Y 65.93, Z 0.00, A 0, B 0, C 0} C_DIS
LIN {X 192.98, Y 66.16, Z 0.00, A 0, B 0, C 0} C_DIS
LIN {X 192.82, Y 66.38, Z 0.00, A 0, B 0, C 0} C_DIS
LIN {X 192.65, Y 66.57, Z 0.00, A 0, B 0, C 0} C_DIS
LIN {X 192.47, Y 66.76, Z 0.00, A 0, B 0, C 0} C_DIS
LIN {X 192.28, Y 66.93, Z 0.00, A 0, B 0, C 0} C_DIS
LIN {X 192.10, Y 67.11, Z 0.00, A 0, B 0, C 0} C_DIS
LIN {X 191.92, Y 67.30, Z 0.00, A 0, B 0, C 0} C_DIS
LIN {X 191.74, Y 67.48, Z 0.00, A 0, B 0, C 0} C_DIS
LIN {X 191.56, Y 67.66, Z 0.00, A 0, B 0, C 0} C_DIS
LIN {X 191.38, Y 67.84, Z 0.00, A 0, B 0, C 0} C_DIS
LIN {X 191.20, Y 68.03, Z 0.00, A 0, B 0, C 0} C_DIS
LIN {X 191.02, Y 68.21, Z 0.00, A 0, B 0, C 0} C_DIS
LIN {X 190.84, Y 68.39, Z 0.00, A 0, B 0, C 0} C_DIS
LIN {X 190.65, Y 68.57, Z 0.00, A 0, B 0, C 0} C_DIS
LIN {X 190.47, Y 68.75, Z 0.00, A 0, B 0, C 0} C_DIS
LIN {X 190.29, Y 68.93, Z 0.00, A 0, B 0, C 0} C_DIS
LIN {X 190.11, Y 69.11, Z 0.00, A 0, B 0, C 0} C_DIS
LIN {X 189.93, Y 69.30, Z 0.00, A 0, B 0, C 0} C_DIS
LIN {X 189.75, Y 69.48, Z 0.00, A 0, B 0, C 0} C_DIS
LIN {X 189.57, Y 69.66, Z 0.00, A 0, B 0, C 0} C_DIS
LIN {X 189.38, Y 69.82, Z 0.00, A 0, B 0, C 0} C_DIS
LIN {X 189.18, Y 69.96, Z 0.00, A 0, B 0, C 0} C_DIS
LIN {X 188.98, Y 70.09, Z 0.00, A 0, B 0, C 0} C_DIS
LIN {X 188.79, Y 70.23, Z 0.00, A 0, B 0, C 0} C_DIS
LIN {X 188.60, Y 70.39, Z 0.00, A 0, B 0, C 0} C_DIS
LIN {X 188.41, Y 70.54, Z 0.00, A 0, B 0, C 0} C_DIS
LIN {X 188.21, Y 70.68, Z 0.00, A 0, B 0, C 0} C_DIS
LIN {X 188.01, Y 70.81, Z 0.00, A 0, B 0, C 0} C_DIS
LIN {X 187.82, Y 70.97, Z 0.00, A 0, B 0, C 0} C_DIS
LIN {X 187.64, Y 71.14, Z 0.00, A 0, B 0, C 0} C_DIS
LIN {X 187.44, Y 71.27, Z 0.00, A 0, B 0, C 0} C_DIS
LIN {X 187.23, Y 71.35, Z 0.00, A 0, B 0, C 0} C_DIS
LIN {X 187.02, Y 71.44, Z 0.00, A 0, B 0, C 0} C_DIS
LIN {X 186.82, Y 71.57, Z 0.00, A 0, B 0, C 0} C_DIS
LIN {X 186.62, Y 71.71, Z 0.00, A 0, B 0, C 0} C_DIS
LIN {X 186.42, Y 71.82, Z 0.00, A 0, B 0, C 0} C_DIS
LIN {X 186.21, Y 71.90, Z 0.00, A 0, B 0, C 0} C_DIS
LIN {X 185.99, Y 71.97, Z 0.00, A 0, B 0, C 0} C_DIS
LIN {X 185.79, Y 72.07, Z 0.00, A 0, B 0, C 0} C_DIS
LIN {X 185.58, Y 72.19, Z 0.00, A 0, B 0, C 0} C_DIS
LIN {X 185.38, Y 72.31, Z 0.00, A 0, B 0, C 0} C_DIS
LIN {X 185.18, Y 72.43, Z 0.00, A 0, B 0, C 0} C_DIS
LIN {X 184.98, Y 72.53, Z 0.00, A 0, B 0, C 0} C_DIS
LIN {X 184.77, Y 72.62, Z 0.00, A 0, B 0, C 0} C_DIS
LIN {X 184.55, Y 72.70, Z 0.00, A 0, B 0, C 0} C_DIS
LIN {X 184.34, Y 72.77, Z 0.00, A 0, B 0, C 0} C_DIS
LIN {X 184.13, Y 72.84, Z 0.00, A 0, B 0, C 0} C_DIS
LIN {X 183.92, Y 72.92, Z 0.00, A 0, B 0, C 0} C_DIS
LIN {X 183.71, Y 73.00, Z 0.00, A 0, B 0, C 0} C_DIS
LIN {X 183.50, Y 73.08, Z 0.00, A 0, B 0, C 0} C_DIS
LIN {X 183.29, Y 73.16, Z 0.00, A 0, B 0, C 0} C_DIS
LIN {X 183.08, Y 73.25, Z 0.00, A 0, B 0, C 0} C_DIS
LIN {X 182.87, Y 73.33, Z 0.00, A 0, B 0, C 0} C_DIS
LIN {X 182.66, Y 73.42, Z 0.00, A 0, B 0, C 0} C_DIS
LIN {X 182.44, Y 73.49, Z 0.00, A 0, B 0, C 0} C_DIS
LIN {X 182.23, Y 73.53, Z 0.00, A 0, B 0, C 0} C_DIS
LIN {X 182.01, Y 73.56, Z 0.00, A 0, B 0, C 0} C_DIS
LIN {X 181.80, Y 73.57, Z 0.00, A 0, B 0, C 0} C_DIS
LIN {X 181.58, Y 73.57, Z 0.00, A 0, B 0, C 0} C_DIS
LIN {X 181.36, Y 73.57, Z 0.00, A 0, B 0, C 0} C_DIS
LIN {X 181.14, Y 73.57, Z 0.00, A 0, B 0, C 0} C_DIS
LIN {X 180.93, Y 73.57, Z 0.00, A 0, B 0, C 0} C_DIS
LIN {X 180.71, Y 73.57, Z 0.00, A 0, B 0, C 0} C_DIS
LIN {X 180.49, Y 73.57, Z 0.00, A 0, B 0, C 0} C_DIS
LIN {X 180.27, Y 73.57, Z 0.00, A 0, B 0, C 0} C_DIS
LIN {X 180.06, Y 73.57, Z 0.00, A 0, B 0, C 0} C_DIS
LIN {X 179.84, Y 73.57, Z 0.00, A 0, B 0, C 0} C_DIS
LIN {X 179.62, Y 73.57, Z 0.00, A 0, B 0, C 0} C_DIS
LIN {X 179.40, Y 73.57, Z 0.00, A 0, B 0, C 0} C_DIS
LIN {X 179.19, Y 73.57, Z 0.00, A 0, B 0, C 0} C_DIS
LIN {X 178.97, Y 73.57, Z 0.00, A 0, B 0, C 0} C_DIS
LIN {X 178.75, Y 73.57, Z 0.00, A 0, B 0, C 0} C_DIS
LIN {X 178.53, Y 73.57, Z 0.00, A 0, B 0, C 0} C_DIS
LIN {X 178.32, Y 73.57, Z 0.00, A 0, B 0, C 0} C_DIS
LIN {X 178.10, Y 73.57, Z 0.00, A 0, B 0, C 0} C_DIS
LIN {X 177.88, Y 73.57, Z 0.00, A 0, B 0, C 0} C_DIS
LIN {X 177.66, Y 73.57, Z 0.00, A 0, B 0, C 0} C_DIS
LIN {X 177.45, Y 73.57, Z 0.00, A 0, B 0, C 0} C_DIS
LIN {X 177.23, Y 73.57, Z 0.00, A 0, B 0, C 0} C_DIS
LIN {X 177.01, Y 73.57, Z 0.00, A 0, B 0, C 0} C_DIS
LIN {X 176.79, Y 73.57, Z 0.00, A 0, B 0, C 0} C_DIS
LIN {X 176.58, Y 73.57, Z 0.00, A 0, B 0, C 0} C_DIS
LIN {X 176.36, Y 73.57, Z 0.00, A 0, B 0, C 0} C_DIS
LIN {X 176.14, Y 73.57, Z 0.00, A 0, B 0, C 0} C_DIS
LIN {X 175.93, Y 73.57, Z 0.00, A 0, B 0, C 0} C_DIS
LIN {X 175.71, Y 73.57, Z 0.00, A 0, B 0, C 0} C_DIS
LIN {X 175.49, Y 73.57, Z 0.00, A 0, B 0, C 0} C_DIS
LIN {X 175.27, Y 73.57, Z 0.00, A 0, B 0, C 0} C_DIS
LIN {X 175.06, Y 73.57, Z 0.00, A 0, B 0, C 0} C_DIS
LIN {X 174.84, Y 73.57, Z 0.00, A 0, B 0, C 0} C_DIS
LIN {X 174.62, Y 73.57, Z 0.00, A 0, B 0, C 0} C_DIS
LIN {X 174.40, Y 73.57, Z 0.00, A 0, B 0, C 0} C_DIS
LIN {X 174.19, Y 73.57, Z 0.00, A 0, B 0, C 0} C_DIS
LIN {X 173.97, Y 73.57, Z 0.00, A 0, B 0, C 0} C_DIS
LIN {X 173.75, Y 73.57, Z 0.00, A 0, B 0, C 0} C_DIS
LIN {X 173.53, Y 73.57, Z 0.00, A 0, B 0, C 0} C_DIS
LIN {X 173.32, Y 73.57, Z 0.00, A 0, B 0, C 0} C_DIS
LIN {X 173.10, Y 73.57, Z 0.00, A 0, B 0, C 0} C_DIS
LIN {X 172.88, Y 73.57, Z 0.00, A 0, B 0, C 0} C_DIS
LIN {X 172.66, Y 73.57, Z 0.00, A 0, B 0, C 0} C_DIS
LIN {X 172.45, Y 73.57, Z 0.00, A 0, B 0, C 0} C_DIS
LIN {X 172.23, Y 73.57, Z 0.00, A 0, B 0, C 0} C_DIS
LIN {X 172.01, Y 73.57, Z 0.00, A 0, B 0, C 0} C_DIS
LIN {X 171.79, Y 73.57, Z 0.00, A 0, B 0, C 0} C_DIS
LIN {X 171.58, Y 73.57, Z 0.00, A 0, B 0, C 0} C_DIS
LIN {X 171.36, Y 73.57, Z 0.00, A 0, B 0, C 0} C_DIS
LIN {X 171.14, Y 73.57, Z 0.00, A 0, B 0, C 0} C_DIS
LIN {X 170.92, Y 73.57, Z 0.00, A 0, B 0, C 0} C_DIS
LIN {X 170.71, Y 73.57, Z 0.00, A 0, B 0, C 0} C_DIS
LIN {X 170.49, Y 73.57, Z 0.00, A 0, B 0, C 0} C_DIS
LIN {X 170.27, Y 73.57, Z 0.00, A 0, B 0, C 0} C_DIS
LIN {X 170.05, Y 73.57, Z 0.00, A 0, B 0, C 0} C_DIS
LIN {X 169.84, Y 73.57, Z 0.00, A 0, B 0, C 0} C_DIS
LIN {X 169.62, Y 73.57, Z 0.00, A 0, B 0, C 0} C_DIS
LIN {X 169.40, Y 73.57, Z 0.00, A 0, B 0, C 0} C_DIS
LIN {X 169.18, Y 73.57, Z 0.00, A 0, B 0, C 0} C_DIS
LIN {X 168.97, Y 73.57, Z 0.00, A 0, B 0, C 0} C_DIS
LIN {X 168.75, Y 73.57, Z 0.00, A 0, B 0, C 0} C_DIS
LIN {X 168.53, Y 73.57, Z 0.00, A 0, B 0, C 0} C_DIS
LIN {X 168.31, Y 73.57, Z 0.00, A 0, B 0, C 0} C_DIS
LIN {X 168.10, Y 73.57, Z 0.00, A 0, B 0, C 0} C_DIS
LIN {X 167.88, Y 73.57, Z 0.00, A 0, B 0, C 0} C_DIS
LIN {X 167.66, Y 73.57, Z 0.00, A 0, B 0, C 0} C_DIS
LIN {X 167.45, Y 73.57, Z 0.00, A 0, B 0, C 0} C_DIS
LIN {X 167.23, Y 73.57, Z 0.00, A 0, B 0, C 0} C_DIS
LIN {X 167.01, Y 73.57, Z 0.00, A 0, B 0, C 0} C_DIS
LIN {X 166.79, Y 73.57, Z 0.00, A 0, B 0, C 0} C_DIS
LIN {X 166.58, Y 73.57, Z 0.00, A 0, B 0, C 0} C_DIS
LIN {X 166.36, Y 73.57, Z 0.00, A 0, B 0, C 0} C_DIS
LIN {X 166.14, Y 73.57, Z 0.00, A 0, B 0, C 0} C_DIS
LIN {X 165.92, Y 73.57, Z 0.00, A 0, B 0, C 0} C_DIS
LIN {X 165.71, Y 73.57, Z 0.00, A 0, B 0, C 0} C_DIS
LIN {X 165.49, Y 73.57, Z 0.00, A 0, B 0, C 0} C_DIS
LIN {X 165.27, Y 73.57, Z 0.00, A 0, B 0, C 0} C_DIS
LIN {X 165.05, Y 73.57, Z 0.00, A 0, B 0, C 0} C_DIS
LIN {X 164.84, Y 73.57, Z 0.00, A 0, B 0, C 0} C_DIS
LIN {X 164.62, Y 73.57, Z 0.00, A 0, B 0, C 0} C_DIS
LIN {X 164.40, Y 73.57, Z 0.00, A 0, B 0, C 0} C_DIS
LIN {X 164.18, Y 73.57, Z 0.00, A 0, B 0, C 0} C_DIS
LIN {X 163.97, Y 73.57, Z 0.00, A 0, B 0, C 0} C_DIS
LIN {X 163.75, Y 73.57, Z 0.00, A 0, B 0, C 0} C_DIS
LIN {X 163.53, Y 73.57, Z 0.00, A 0, B 0, C 0} C_DIS
LIN {X 163.31, Y 73.57, Z 0.00, A 0, B 0, C 0} C_DIS
LIN {X 163.10, Y 73.57, Z 0.00, A 0, B 0, C 0} C_DIS
LIN {X 162.88, Y 73.57, Z 0.00, A 0, B 0, C 0} C_DIS
LIN {X 162.66, Y 73.57, Z 0.00, A 0, B 0, C 0} C_DIS
LIN {X 162.44, Y 73.57, Z 0.00, A 0, B 0, C 0} C_DIS
LIN {X 162.23, Y 73.57, Z 0.00, A 0, B 0, C 0} C_DIS
LIN {X 162.01, Y 73.57, Z 0.00, A 0, B 0, C 0} C_DIS
LIN {X 161.79, Y 73.57, Z 0.00, A 0, B 0, C 0} C_DIS
LIN {X 161.57, Y 73.57, Z 0.00, A 0, B 0, C 0} C_DIS
LIN {X 161.36, Y 73.57, Z 0.00, A 0, B 0, C 0} C_DIS
LIN {X 161.14, Y 73.57, Z 0.00, A 0, B 0, C 0} C_DIS
LIN {X 160.92, Y 73.57, Z 0.00, A 0, B 0, C 0} C_DIS
LIN {X 160.70, Y 73.57, Z 0.00, A 0, B 0, C 0} C_DIS
LIN {X 160.49, Y 73.57, Z 0.00, A 0, B 0, C 0} C_DIS
LIN {X 160.27, Y 73.57, Z 0.00, A 0, B 0, C 0} C_DIS
LIN {X 160.05, Y 73.57, Z 0.00, A 0, B 0, C 0} C_DIS
LIN {X 159.84, Y 73.56, Z 0.00, A 0, B 0, C 0} C_DIS
LIN {X 159.62, Y 73.56, Z 0.00, A 0, B 0, C 0} C_DIS
LIN {X 159.40, Y 73.56, Z 0.00, A 0, B 0, C 0} C_DIS
LIN {X 159.18, Y 73.56, Z 0.00, A 0, B 0, C 0} C_DIS
LIN {X 158.97, Y 73.56, Z 0.00, A 0, B 0, C 0} C_DIS
LIN {X 158.75, Y 73.56, Z 0.00, A 0, B 0, C 0} C_DIS
LIN {X 158.53, Y 73.57, Z 0.00, A 0, B 0, C 0} C_DIS
LIN {X 158.31, Y 73.57, Z 0.00, A 0, B 0, C 0} C_DIS
LIN {X 158.09, Y 73.58, Z 0.00, A 0, B 0, C 0} C_DIS
LIN {X 157.88, Y 73.58, Z 0.00, A 0, B 0, C 0} C_DIS
LIN {X 157.66, Y 73.58, Z 0.00, A 0, B 0, C 0} C_DIS
LIN {X 157.44, Y 73.58, Z 0.00, A 0, B 0, C 0} C_DIS
LIN {X 157.23, Y 73.57, Z 0.00, A 0, B 0, C 0} C_DIS
LIN {X 157.01, Y 73.54, Z 0.00, A 0, B 0, C 0} C_DIS
LIN {X 156.80, Y 73.49, Z 0.00, A 0, B 0, C 0} C_DIS
LIN {X 156.58, Y 73.43, Z 0.00, A 0, B 0, C 0} C_DIS
LIN {X 156.37, Y 73.36, Z 0.00, A 0, B 0, C 0} C_DIS
LIN {X 156.16, Y 73.29, Z 0.00, A 0, B 0, C 0} C_DIS
LIN {X 155.95, Y 73.20, Z 0.00, A 0, B 0, C 0} C_DIS
LIN {X 155.74, Y 73.12, Z 0.00, A 0, B 0, C 0} C_DIS
LIN {X 155.53, Y 73.03, Z 0.00, A 0, B 0, C 0} C_DIS
LIN {X 155.32, Y 72.95, Z 0.00, A 0, B 0, C 0} C_DIS
LIN {X 155.11, Y 72.87, Z 0.00, A 0, B 0, C 0} C_DIS
LIN {X 154.89, Y 72.80, Z 0.00, A 0, B 0, C 0} C_DIS
LIN {X 154.68, Y 72.73, Z 0.00, A 0, B 0, C 0} C_DIS
LIN {X 154.47, Y 72.65, Z 0.00, A 0, B 0, C 0} C_DIS
LIN {X 154.26, Y 72.54, Z 0.00, A 0, B 0, C 0} C_DIS
LIN {X 154.07, Y 72.40, Z 0.00, A 0, B 0, C 0} C_DIS
LIN {X 153.89, Y 72.23, Z 0.00, A 0, B 0, C 0} C_DIS
LIN {X 153.69, Y 72.08, Z 0.00, A 0, B 0, C 0} C_DIS
LIN {X 153.49, Y 71.95, Z 0.00, A 0, B 0, C 0} C_DIS
LIN {X 153.29, Y 71.82, Z 0.00, A 0, B 0, C 0} C_DIS
LIN {X 153.10, Y 71.66, Z 0.00, A 0, B 0, C 0} C_DIS
LIN {X 152.92, Y 71.49, Z 0.00, A 0, B 0, C 0} C_DIS
LIN {X 152.74, Y 71.30, Z 0.00, A 0, B 0, C 0} C_DIS
LIN {X 152.56, Y 71.12, Z 0.00, A 0, B 0, C 0} C_DIS
LIN {X 152.38, Y 70.93, Z 0.00, A 0, B 0, C 0} C_DIS
LIN {X 152.20, Y 70.75, Z 0.00, A 0, B 0, C 0} C_DIS
LIN {X 152.02, Y 70.57, Z 0.00, A 0, B 0, C 0} C_DIS
LIN {X 151.83, Y 70.40, Z 0.00, A 0, B 0, C 0} C_DIS
LIN {X 151.65, Y 70.22, Z 0.00, A 0, B 0, C 0} C_DIS
LIN {X 151.47, Y 70.03, Z 0.00, A 0, B 0, C 0} C_DIS
LIN {X 151.30, Y 69.84, Z 0.00, A 0, B 0, C 0} C_DIS
LIN {X 151.12, Y 69.64, Z 0.00, A 0, B 0, C 0} C_DIS
LIN {X 150.96, Y 69.43, Z 0.00, A 0, B 0, C 0} C_DIS
LIN {X 150.80, Y 69.21, Z 0.00, A 0, B 0, C 0} C_DIS
LIN {X 150.65, Y 68.98, Z 0.00, A 0, B 0, C 0} C_DIS
LIN {X 150.50, Y 68.74, Z 0.00, A 0, B 0, C 0} C_DIS
LIN {X 150.35, Y 68.50, Z 0.00, A 0, B 0, C 0} C_DIS
LIN {X 150.19, Y 68.27, Z 0.00, A 0, B 0, C 0} C_DIS
LIN {X 150.03, Y 68.04, Z 0.00, A 0, B 0, C 0} C_DIS
LIN {X 149.88, Y 67.82, Z 0.00, A 0, B 0, C 0} C_DIS
LIN {X 149.73, Y 67.58, Z 0.00, A 0, B 0, C 0} C_DIS
LIN {X 149.59, Y 67.33, Z 0.00, A 0, B 0, C 0} C_DIS
LIN {X 149.46, Y 67.07, Z 0.00, A 0, B 0, C 0} C_DIS
LIN {X 149.34, Y 66.80, Z 0.00, A 0, B 0, C 0} C_DIS
LIN {X 149.21, Y 66.53, Z 0.00, A 0, B 0, C 0} C_DIS
LIN {X 149.10, Y 66.25, Z 0.00, A 0, B 0, C 0} C_DIS
LIN {X 148.98, Y 65.98, Z 0.00, A 0, B 0, C 0} C_DIS
LIN {X 148.86, Y 65.70, Z 0.00, A 0, B 0, C 0} C_DIS
LIN {X 148.74, Y 65.43, Z 0.00, A 0, B 0, C 0} C_DIS
LIN {X 148.62, Y 65.16, Z 0.00, A 0, B 0, C 0} C_DIS
LIN {X 148.49, Y 64.89, Z 0.00, A 0, B 0, C 0} C_DIS
LIN {X 148.37, Y 64.62, Z 0.00, A 0, B 0, C 0} C_DIS
LIN {X 148.25, Y 64.34, Z 0.00, A 0, B 0, C 0} C_DIS
LIN {X 148.16, Y 64.05, Z 0.00, A 0, B 0, C 0} C_DIS
LIN {X 148.08, Y 63.74, Z 0.00, A 0, B 0, C 0} C_DIS
LIN {X 147.98, Y 63.45, Z 0.00, A 0, B 0, C 0} C_DIS
LIN {X 147.86, Y 63.18, Z 0.00, A 0, B 0, C 0} C_DIS
LIN {X 147.71, Y 62.95, Z 0.00, A 0, B 0, C 0} C_DIS
LIN {X 147.55, Y 62.72, Z 0.00, A 0, B 0, C 0} C_DIS
LIN {X 147.40, Y 62.49, Z 0.00, A 0, B 0, C 0} C_DIS
LIN {X 147.23, Y 62.29, Z 0.00, A 0, B 0, C 0} C_DIS
LIN {X 147.04, Y 62.14, Z 0.00, A 0, B 0, C 0} C_DIS
LIN {X 146.83, Y 62.04, Z 0.00, A 0, B 0, C 0} C_DIS
LIN {X 146.62, Y 61.97, Z 0.00, A 0, B 0, C 0} C_DIS
LIN {X 146.40, Y 61.90, Z 0.00, A 0, B 0, C 0} C_DIS
LIN {X 146.19, Y 61.84, Z 0.00, A 0, B 0, C 0} C_DIS
LIN {X 145.98, Y 61.80, Z 0.00, A 0, B 0, C 0} C_DIS
LIN {X 145.76, Y 61.77, Z 0.00, A 0, B 0, C 0} C_DIS
LIN {X 145.54, Y 61.76, Z 0.00, A 0, B 0, C 0} C_DIS
LIN {X 145.33, Y 61.76, Z 0.00, A 0, B 0, C 0} C_DIS
LIN {X 145.11, Y 61.76, Z 0.00, A 0, B 0, C 0} C_DIS
LIN {X 144.89, Y 61.77, Z 0.00, A 0, B 0, C 0} C_DIS
LIN {X 144.67, Y 61.77, Z 0.00, A 0, B 0, C 0} C_DIS
LIN {X 144.45, Y 61.78, Z 0.00, A 0, B 0, C 0} C_DIS
LIN {X 144.24, Y 61.78, Z 0.00, A 0, B 0, C 0} C_DIS
LIN {X 144.02, Y 61.78, Z 0.00, A 0, B 0, C 0} C_DIS
LIN {X 143.80, Y 61.78, Z 0.00, A 0, B 0, C 0} C_DIS
LIN {X 143.59, Y 61.78, Z 0.00, A 0, B 0, C 0} C_DIS
LIN {X 143.37, Y 61.77, Z 0.00, A 0, B 0, C 0} C_DIS
LIN {X 143.15, Y 61.77, Z 0.00, A 0, B 0, C 0} C_DIS
LIN {X 142.93, Y 61.76, Z 0.00, A 0, B 0, C 0} C_DIS
LIN {X 142.72, Y 61.76, Z 0.00, A 0, B 0, C 0} C_DIS
LIN {X 142.50, Y 61.76, Z 0.00, A 0, B 0, C 0} C_DIS
LIN {X 142.28, Y 61.76, Z 0.00, A 0, B 0, C 0} C_DIS
LIN {X 142.06, Y 61.78, Z 0.00, A 0, B 0, C 0} C_DIS
LIN {X 141.85, Y 61.80, Z 0.00, A 0, B 0, C 0} C_DIS
LIN {X 141.63, Y 61.84, Z 0.00, A 0, B 0, C 0} C_DIS
LIN {X 141.42, Y 61.89, Z 0.00, A 0, B 0, C 0} C_DIS
LIN {X 141.21, Y 61.97, Z 0.00, A 0, B 0, C 0} C_DIS
LIN {X 140.99, Y 62.05, Z 0.00, A 0, B 0, C 0} C_DIS
LIN {X 140.79, Y 62.16, Z 0.00, A 0, B 0, C 0} C_DIS
LIN {X 140.59, Y 62.29, Z 0.00, A 0, B 0, C 0} C_DIS
LIN {X 140.43, Y 62.49, Z 0.00, A 0, B 0, C 0} C_DIS
LIN {X 140.27, Y 62.73, Z 0.00, A 0, B 0, C 0} C_DIS
LIN {X 140.12, Y 62.97, Z 0.00, A 0, B 0, C 0} C_DIS
LIN {X 139.96, Y 63.20, Z 0.00, A 0, B 0, C 0} C_DIS
LIN {X 139.84, Y 63.46, Z 0.00, A 0, B 0, C 0} C_DIS
LIN {X 139.76, Y 63.76, Z 0.00, A 0, B 0, C 0} C_DIS
LIN {X 139.70, Y 64.08, Z 0.00, A 0, B 0, C 0} C_DIS
LIN {X 139.65, Y 64.40, Z 0.00, A 0, B 0, C 0} C_DIS
LIN {X 139.59, Y 64.72, Z 0.00, A 0, B 0, C 0} C_DIS
LIN {X 139.57, Y 65.04, Z 0.00, A 0, B 0, C 0} C_DIS
LIN {X 139.58, Y 65.36, Z 0.00, A 0, B 0, C 0} C_DIS
LIN {X 139.62, Y 65.69, Z 0.00, A 0, B 0, C 0} C_DIS
LIN {X 139.67, Y 66.01, Z 0.00, A 0, B 0, C 0} C_DIS
LIN {X 139.72, Y 66.33, Z 0.00, A 0, B 0, C 0} C_DIS
LIN {X 139.80, Y 66.63, Z 0.00, A 0, B 0, C 0} C_DIS
LIN {X 139.91, Y 66.92, Z 0.00, A 0, B 0, C 0} C_DIS
LIN {X 140.02, Y 67.20, Z 0.00, A 0, B 0, C 0} C_DIS
LIN {X 140.11, Y 67.49, Z 0.00, A 0, B 0, C 0} C_DIS
LIN {X 140.20, Y 67.79, Z 0.00, A 0, B 0, C 0} C_DIS
LIN {X 140.29, Y 68.09, Z 0.00, A 0, B 0, C 0} C_DIS
LIN {X 140.40, Y 68.37, Z 0.00, A 0, B 0, C 0} C_DIS
LIN {X 140.50, Y 68.66, Z 0.00, A 0, B 0, C 0} C_DIS
LIN {X 140.59, Y 68.96, Z 0.00, A 0, B 0, C 0} C_DIS
LIN {X 140.68, Y 69.26, Z 0.00, A 0, B 0, C 0} C_DIS
LIN {X 140.78, Y 69.54, Z 0.00, A 0, B 0, C 0} C_DIS
LIN {X 140.89, Y 69.83, Z 0.00, A 0, B 0, C 0} C_DIS
LIN {X 140.98, Y 70.13, Z 0.00, A 0, B 0, C 0} C_DIS
LIN {X 141.07, Y 70.43, Z 0.00, A 0, B 0, C 0} C_DIS
LIN {X 141.16, Y 70.72, Z 0.00, A 0, B 0, C 0} C_DIS
LIN {X 141.27, Y 71.00, Z 0.00, A 0, B 0, C 0} C_DIS
LIN {X 141.39, Y 71.28, Z 0.00, A 0, B 0, C 0} C_DIS
LIN {X 141.51, Y 71.55, Z 0.00, A 0, B 0, C 0} C_DIS
LIN {X 141.63, Y 71.82, Z 0.00, A 0, B 0, C 0} C_DIS
LIN {X 141.75, Y 72.10, Z 0.00, A 0, B 0, C 0} C_DIS
LIN {X 141.87, Y 72.37, Z 0.00, A 0, B 0, C 0} C_DIS
LIN {X 141.99, Y 72.64, Z 0.00, A 0, B 0, C 0} C_DIS
LIN {X 142.11, Y 72.91, Z 0.00, A 0, B 0, C 0} C_DIS
LIN {X 142.23, Y 73.19, Z 0.00, A 0, B 0, C 0} C_DIS
LIN {X 142.35, Y 73.46, Z 0.00, A 0, B 0, C 0} C_DIS
LIN {X 142.48, Y 73.73, Z 0.00, A 0, B 0, C 0} C_DIS
LIN {X 142.61, Y 73.99, Z 0.00, A 0, B 0, C 0} C_DIS
LIN {X 142.75, Y 74.24, Z 0.00, A 0, B 0, C 0} C_DIS
LIN {X 142.90, Y 74.47, Z 0.00, A 0, B 0, C 0} C_DIS
LIN {X 143.05, Y 74.70, Z 0.00, A 0, B 0, C 0} C_DIS
LIN {X 143.21, Y 74.93, Z 0.00, A 0, B 0, C 0} C_DIS
LIN {X 143.36, Y 75.16, Z 0.00, A 0, B 0, C 0} C_DIS
LIN {X 143.51, Y 75.41, Z 0.00, A 0, B 0, C 0} C_DIS
LIN {X 143.63, Y 75.67, Z 0.00, A 0, B 0, C 0} C_DIS
LIN {X 143.75, Y 75.95, Z 0.00, A 0, B 0, C 0} C_DIS
LIN {X 143.88, Y 76.21, Z 0.00, A 0, B 0, C 0} C_DIS
LIN {X 144.03, Y 76.44, Z 0.00, A 0, B 0, C 0} C_DIS
LIN {X 144.19, Y 76.68, Z 0.00, A 0, B 0, C 0} C_DIS
LIN {X 144.34, Y 76.90, Z 0.00, A 0, B 0, C 0} C_DIS
LIN {X 144.51, Y 77.11, Z 0.00, A 0, B 0, C 0} C_DIS
LIN {X 144.69, Y 77.30, Z 0.00, A 0, B 0, C 0} C_DIS
LIN {X 144.86, Y 77.49, Z 0.00, A 0, B 0, C 0} C_DIS
LIN {X 145.03, Y 77.69, Z 0.00, A 0, B 0, C 0} C_DIS
LIN {X 145.20, Y 77.90, Z 0.00, A 0, B 0, C 0} C_DIS
LIN {X 145.35, Y 78.14, Z 0.00, A 0, B 0, C 0} C_DIS
LIN {X 145.50, Y 78.38, Z 0.00, A 0, B 0, C 0} C_DIS
LIN {X 145.65, Y 78.62, Z 0.00, A 0, B 0, C 0} C_DIS
LIN {X 145.80, Y 78.85, Z 0.00, A 0, B 0, C 0} C_DIS
LIN {X 145.96, Y 79.07, Z 0.00, A 0, B 0, C 0} C_DIS
LIN {X 146.12, Y 79.29, Z 0.00, A 0, B 0, C 0} C_DIS
LIN {X 146.27, Y 79.52, Z 0.00, A 0, B 0, C 0} C_DIS
LIN {X 146.42, Y 79.77, Z 0.00, A 0, B 0, C 0} C_DIS
LIN {X 146.56, Y 80.03, Z 0.00, A 0, B 0, C 0} C_DIS
LIN {X 146.68, Y 80.31, Z 0.00, A 0, B 0, C 0} C_DIS
LIN {X 146.77, Y 80.61, Z 0.00, A 0, B 0, C 0} C_DIS
LIN {X 146.84, Y 80.91, Z 0.00, A 0, B 0, C 0} C_DIS
LIN {X 146.88, Y 81.22, Z 0.00, A 0, B 0, C 0} C_DIS
LIN {X 146.90, Y 81.54, Z 0.00, A 0, B 0, C 0} C_DIS
LIN {X 146.92, Y 81.87, Z 0.00, A 0, B 0, C 0} C_DIS
LIN {X 146.92, Y 82.20, Z 0.00, A 0, B 0, C 0} C_DIS
LIN {X 146.92, Y 82.52, Z 0.00, A 0, B 0, C 0} C_DIS
LIN {X 146.92, Y 82.85, Z 0.00, A 0, B 0, C 0} C_DIS
LIN {X 146.92, Y 83.18, Z 0.00, A 0, B 0, C 0} C_DIS
LIN {X 146.92, Y 83.51, Z 0.00, A 0, B 0, C 0} C_DIS
LIN {X 146.92, Y 83.84, Z 0.00, A 0, B 0, C 0} C_DIS
LIN {X 146.92, Y 84.17, Z 0.00, A 0, B 0, C 0} C_DIS
LIN {X 146.92, Y 84.50, Z 0.00, A 0, B 0, C 0} C_DIS
LIN {X 146.92, Y 84.83, Z 0.00, A 0, B 0, C 0} C_DIS
LIN {X 146.92, Y 85.16, Z 0.00, A 0, B 0, C 0} C_DIS
LIN {X 146.92, Y 85.48, Z 0.00, A 0, B 0, C 0} C_DIS
LIN {X 146.92, Y 85.81, Z 0.00, A 0, B 0, C 0} C_DIS
LIN {X 146.92, Y 86.14, Z 0.00, A 0, B 0, C 0} C_DIS
LIN {X 146.92, Y 86.47, Z 0.00, A 0, B 0, C 0} C_DIS
LIN {X 146.92, Y 86.80, Z 0.00, A 0, B 0, C 0} C_DIS
LIN {X 146.92, Y 87.12, Z 0.00, A 0, B 0, C 0} C_DIS
LIN {X 146.92, Y 87.45, Z 0.00, A 0, B 0, C 0} C_DIS
LIN {X 146.92, Y 87.78, Z 0.00, A 0, B 0, C 0} C_DIS
LIN {X 146.92, Y 88.11, Z 0.00, A 0, B 0, C 0} C_DIS
LIN {X 146.92, Y 88.44, Z 0.00, A 0, B 0, C 0} C_DIS
LIN {X 146.92, Y 88.76, Z 0.00, A 0, B 0, C 0} C_DIS
LIN {X 146.92, Y 89.09, Z 0.00, A 0, B 0, C 0} C_DIS
LIN {X 146.92, Y 89.42, Z 0.00, A 0, B 0, C 0} C_DIS
LIN {X 146.92, Y 89.75, Z 0.00, A 0, B 0, C 0} C_DIS
LIN {X 146.92, Y 90.07, Z 0.00, A 0, B 0, C 0} C_DIS
LIN {X 146.92, Y 90.40, Z 0.00, A 0, B 0, C 0} C_DIS
LIN {X 146.92, Y 90.73, Z 0.00, A 0, B 0, C 0} C_DIS
LIN {X 146.92, Y 91.06, Z 0.00, A 0, B 0, C 0} C_DIS
LIN {X 146.92, Y 91.38, Z 0.00, A 0, B 0, C 0} C_DIS
LIN {X 146.92, Y 91.71, Z 0.00, A 0, B 0, C 0} C_DIS
LIN {X 146.92, Y 92.04, Z 0.00, A 0, B 0, C 0} C_DIS
LIN {X 146.92, Y 92.36, Z 0.00, A 0, B 0, C 0} C_DIS
LIN {X 146.92, Y 92.69, Z 0.00, A 0, B 0, C 0} C_DIS
LIN {X 146.92, Y 93.02, Z 0.00, A 0, B 0, C 0} C_DIS
LIN {X 146.92, Y 93.35, Z 0.00, A 0, B 0, C 0} C_DIS
LIN {X 146.92, Y 93.67, Z 0.00, A 0, B 0, C 0} C_DIS
LIN {X 146.92, Y 94.00, Z 0.00, A 0, B 0, C 0} C_DIS
LIN {X 146.92, Y 94.33, Z 0.00, A 0, B 0, C 0} C_DIS
LIN {X 146.92, Y 94.66, Z 0.00, A 0, B 0, C 0} C_DIS
LIN {X 146.92, Y 94.98, Z 0.00, A 0, B 0, C 0} C_DIS
LIN {X 146.92, Y 95.31, Z 0.00, A 0, B 0, C 0} C_DIS
LIN {X 146.92, Y 95.64, Z 0.00, A 0, B 0, C 0} C_DIS
LIN {X 146.92, Y 95.97, Z 0.00, A 0, B 0, C 0} C_DIS
LIN {X 146.92, Y 96.30, Z 0.00, A 0, B 0, C 0} C_DIS
LIN {X 146.92, Y 96.62, Z 0.00, A 0, B 0, C 0} C_DIS
LIN {X 146.92, Y 96.95, Z 0.00, A 0, B 0, C 0} C_DIS
LIN {X 146.92, Y 97.28, Z 0.00, A 0, B 0, C 0} C_DIS
LIN {X 146.92, Y 97.61, Z 0.00, A 0, B 0, C 0} C_DIS
LIN {X 146.92, Y 97.93, Z 0.00, A 0, B 0, C 0} C_DIS
LIN {X 146.92, Y 98.26, Z 0.00, A 0, B 0, C 0} C_DIS
LIN {X 146.92, Y 98.59, Z 0.00, A 0, B 0, C 0} C_DIS
LIN {X 146.92, Y 98.92, Z 0.00, A 0, B 0, C 0} C_DIS
LIN {X 146.92, Y 99.25, Z 0.00, A 0, B 0, C 0} C_DIS
LIN {X 146.92, Y 99.57, Z 0.00, A 0, B 0, C 0} C_DIS
LIN {X 146.92, Y 99.90, Z 0.00, A 0, B 0, C 0} C_DIS
LIN {X 146.92, Y 100.23, Z 0.00, A 0, B 0, C 0} C_DIS
LIN {X 146.92, Y 100.56, Z 0.00, A 0, B 0, C 0} C_DIS
LIN {X 146.92, Y 100.88, Z 0.00, A 0, B 0, C 0} C_DIS
LIN {X 146.92, Y 101.21, Z 0.00, A 0, B 0, C 0} C_DIS
LIN {X 146.92, Y 101.54, Z 0.00, A 0, B 0, C 0} C_DIS
LIN {X 146.92, Y 101.87, Z 0.00, A 0, B 0, C 0} C_DIS
LIN {X 146.92, Y 102.20, Z 0.00, A 0, B 0, C 0} C_DIS
LIN {X 146.92, Y 102.52, Z 0.00, A 0, B 0, C 0} C_DIS
LIN {X 146.92, Y 102.85, Z 0.00, A 0, B 0, C 0} C_DIS
LIN {X 146.92, Y 103.18, Z 0.00, A 0, B 0, C 0} C_DIS
LIN {X 146.92, Y 103.51, Z 0.00, A 0, B 0, C 0} C_DIS
LIN {X 146.92, Y 103.83, Z 0.00, A 0, B 0, C 0} C_DIS
LIN {X 146.92, Y 104.16, Z 0.00, A 0, B 0, C 0} C_DIS
LIN {X 146.92, Y 104.49, Z 0.00, A 0, B 0, C 0} C_DIS
LIN {X 146.92, Y 104.82, Z 0.00, A 0, B 0, C 0} C_DIS
LIN {X 146.92, Y 105.15, Z 0.00, A 0, B 0, C 0} C_DIS
LIN {X 146.92, Y 105.47, Z 0.00, A 0, B 0, C 0} C_DIS
LIN {X 146.92, Y 105.80, Z 0.00, A 0, B 0, C 0} C_DIS
LIN {X 146.92, Y 106.13, Z 0.00, A 0, B 0, C 0} C_DIS
LIN {X 146.92, Y 106.46, Z 0.00, A 0, B 0, C 0} C_DIS
LIN {X 146.92, Y 106.78, Z 0.00, A 0, B 0, C 0} C_DIS
LIN {X 146.92, Y 107.11, Z 0.00, A 0, B 0, C 0} C_DIS
LIN {X 146.92, Y 107.44, Z 0.00, A 0, B 0, C 0} C_DIS
LIN {X 146.92, Y 107.77, Z 0.00, A 0, B 0, C 0} C_DIS
LIN {X 146.92, Y 108.09, Z 0.00, A 0, B 0, C 0} C_DIS
LIN {X 146.92, Y 108.42, Z 0.00, A 0, B 0, C 0} C_DIS
LIN {X 146.92, Y 108.75, Z 0.00, A 0, B 0, C 0} C_DIS
LIN {X 146.92, Y 109.08, Z 0.00, A 0, B 0, C 0} C_DIS
LIN {X 146.92, Y 109.40, Z 0.00, A 0, B 0, C 0} C_DIS
LIN {X 146.92, Y 109.73, Z 0.00, A 0, B 0, C 0} C_DIS
LIN {X 146.92, Y 110.06, Z 0.00, A 0, B 0, C 0} C_DIS
LIN {X 146.92, Y 110.39, Z 0.00, A 0, B 0, C 0} C_DIS
LIN {X 146.92, Y 110.71, Z 0.00, A 0, B 0, C 0} C_DIS
LIN {X 146.92, Y 111.04, Z 0.00, A 0, B 0, C 0} C_DIS
LIN {X 146.92, Y 111.37, Z 0.00, A 0, B 0, C 0} C_DIS
LIN {X 146.92, Y 111.70, Z 0.00, A 0, B 0, C 0} C_DIS
LIN {X 146.92, Y 112.03, Z 0.00, A 0, B 0, C 0} C_DIS
LIN {X 146.92, Y 112.35, Z 0.00, A 0, B 0, C 0} C_DIS
LIN {X 146.92, Y 112.68, Z 0.00, A 0, B 0, C 0} C_DIS
LIN {X 146.92, Y 113.01, Z 0.00, A 0, B 0, C 0} C_DIS
LIN {X 146.92, Y 113.34, Z 0.00, A 0, B 0, C 0} C_DIS
LIN {X 146.92, Y 113.67, Z 0.00, A 0, B 0, C 0} C_DIS
LIN {X 146.92, Y 113.99, Z 0.00, A 0, B 0, C 0} C_DIS
LIN {X 146.92, Y 114.32, Z 0.00, A 0, B 0, C 0} C_DIS
LIN {X 146.92, Y 114.65, Z 0.00, A 0, B 0, C 0} C_DIS
LIN {X 146.92, Y 114.97, Z 0.00, A 0, B 0, C 0} C_DIS
LIN {X 146.93, Y 115.30, Z 0.00, A 0, B 0, C 0} C_DIS
LIN {X 146.95, Y 115.63, Z 0.00, A 0, B 0, C 0} C_DIS
LIN {X 146.98, Y 115.95, Z 0.00, A 0, B 0, C 0} C_DIS
LIN {X 147.03, Y 116.27, Z 0.00, A 0, B 0, C 0} C_DIS
LIN {X 147.08, Y 116.59, Z 0.00, A 0, B 0, C 0} C_DIS
LIN {X 147.15, Y 116.90, Z 0.00, A 0, B 0, C 0} C_DIS
LIN {X 147.23, Y 117.21, Z 0.00, A 0, B 0, C 0} C_DIS
LIN {X 147.34, Y 117.48, Z 0.00, A 0, B 0, C 0} C_DIS
LIN {X 147.49, Y 117.71, Z 0.00, A 0, B 0, C 0} C_DIS
LIN {X 147.65, Y 117.95, Z 0.00, A 0, B 0, C 0} C_DIS
LIN {X 147.81, Y 118.17, Z 0.00, A 0, B 0, C 0} C_DIS
LIN {X 147.98, Y 118.38, Z 0.00, A 0, B 0, C 0} C_DIS
LIN {X 148.15, Y 118.57, Z 0.00, A 0, B 0, C 0} C_DIS
LIN {X 148.32, Y 118.77, Z 0.00, A 0, B 0, C 0} C_DIS
LIN {X 148.49, Y 118.97, Z 0.00, A 0, B 0, C 0} C_DIS
LIN {X 148.66, Y 119.18, Z 0.00, A 0, B 0, C 0} C_DIS
LIN {X 148.82, Y 119.40, Z 0.00, A 0, B 0, C 0} C_DIS
LIN {X 148.97, Y 119.64, Z 0.00, A 0, B 0, C 0} C_DIS
LIN {X 149.12, Y 119.88, Z 0.00, A 0, B 0, C 0} C_DIS
LIN {X 149.27, Y 120.12, Z 0.00, A 0, B 0, C 0} C_DIS
LIN {X 149.42, Y 120.35, Z 0.00, A 0, B 0, C 0} C_DIS
LIN {X 149.58, Y 120.58, Z 0.00, A 0, B 0, C 0} C_DIS
LIN {X 149.74, Y 120.80, Z 0.00, A 0, B 0, C 0} C_DIS
LIN {X 149.91, Y 121.00, Z 0.00, A 0, B 0, C 0} C_DIS
LIN {X 150.08, Y 121.19, Z 0.00, A 0, B 0, C 0} C_DIS
LIN {X 150.26, Y 121.37, Z 0.00, A 0, B 0, C 0} C_DIS
LIN {X 150.45, Y 121.54, Z 0.00, A 0, B 0, C 0} C_DIS
LIN {X 150.64, Y 121.71, Z 0.00, A 0, B 0, C 0} C_DIS
LIN {X 150.82, Y 121.89, Z 0.00, A 0, B 0, C 0} C_DIS
LIN {X 150.99, Y 122.09, Z 0.00, A 0, B 0, C 0} C_DIS
LIN {X 151.15, Y 122.31, Z 0.00, A 0, B 0, C 0} C_DIS
LIN {X 151.31, Y 122.54, Z 0.00, A 0, B 0, C 0} C_DIS
LIN {X 151.46, Y 122.77, Z 0.00, A 0, B 0, C 0} C_DIS
LIN {X 151.62, Y 123.00, Z 0.00, A 0, B 0, C 0} C_DIS
LIN {X 151.77, Y 123.22, Z 0.00, A 0, B 0, C 0} C_DIS
LIN {X 151.93, Y 123.46, Z 0.00, A 0, B 0, C 0} C_DIS
LIN {X 152.08, Y 123.69, Z 0.00, A 0, B 0, C 0} C_DIS
LIN {X 152.24, Y 123.92, Z 0.00, A 0, B 0, C 0} C_DIS
LIN {X 152.39, Y 124.15, Z 0.00, A 0, B 0, C 0} C_DIS
LIN {X 152.54, Y 124.38, Z 0.00, A 0, B 0, C 0} C_DIS
LIN {X 152.70, Y 124.62, Z 0.00, A 0, B 0, C 0} C_DIS
LIN {X 152.85, Y 124.85, Z 0.00, A 0, B 0, C 0} C_DIS
LIN {X 153.00, Y 125.08, Z 0.00, A 0, B 0, C 0} C_DIS
LIN {X 153.16, Y 125.31, Z 0.00, A 0, B 0, C 0} C_DIS
LIN {X 153.31, Y 125.55, Z 0.00, A 0, B 0, C 0} C_DIS
LIN {X 153.46, Y 125.78, Z 0.00, A 0, B 0, C 0} C_DIS
LIN {X 153.62, Y 126.01, Z 0.00, A 0, B 0, C 0} C_DIS
LIN {X 153.77, Y 126.24, Z 0.00, A 0, B 0, C 0} C_DIS
LIN {X 153.92, Y 126.47, Z 0.00, A 0, B 0, C 0} C_DIS
LIN {X 154.08, Y 126.70, Z 0.00, A 0, B 0, C 0} C_DIS
LIN {X 154.23, Y 126.93, Z 0.00, A 0, B 0, C 0} C_DIS
LIN {X 154.39, Y 127.17, Z 0.00, A 0, B 0, C 0} C_DIS
LIN {X 154.54, Y 127.40, Z 0.00, A 0, B 0, C 0} C_DIS
LIN {X 154.70, Y 127.63, Z 0.00, A 0, B 0, C 0} C_DIS
LIN {X 154.85, Y 127.86, Z 0.00, A 0, B 0, C 0} C_DIS
LIN {X 155.00, Y 128.09, Z 0.00, A 0, B 0, C 0} C_DIS
LIN {X 155.16, Y 128.32, Z 0.00, A 0, B 0, C 0} C_DIS
LIN {X 155.31, Y 128.56, Z 0.00, A 0, B 0, C 0} C_DIS
LIN {X 155.46, Y 128.79, Z 0.00, A 0, B 0, C 0} C_DIS
LIN {X 155.61, Y 129.03, Z 0.00, A 0, B 0, C 0} C_DIS
LIN {X 155.75, Y 129.28, Z 0.00, A 0, B 0, C 0} C_DIS
LIN {X 155.87, Y 129.55, Z 0.00, A 0, B 0, C 0} C_DIS
LIN {X 155.98, Y 129.83, Z 0.00, A 0, B 0, C 0} C_DIS
LIN {X 156.10, Y 130.11, Z 0.00, A 0, B 0, C 0} C_DIS
LIN {X 156.22, Y 130.39, Z 0.00, A 0, B 0, C 0} C_DIS
LIN {X 156.34, Y 130.65, Z 0.00, A 0, B 0, C 0} C_DIS
LIN {X 156.47, Y 130.92, Z 0.00, A 0, B 0, C 0} C_DIS
LIN {X 156.61, Y 131.17, Z 0.00, A 0, B 0, C 0} C_DIS
LIN {X 156.76, Y 131.41, Z 0.00, A 0, B 0, C 0} C_DIS
LIN {X 156.91, Y 131.64, Z 0.00, A 0, B 0, C 0} C_DIS
LIN {X 157.07, Y 131.86, Z 0.00, A 0, B 0, C 0} C_DIS
LIN {X 157.23, Y 132.09, Z 0.00, A 0, B 0, C 0} C_DIS
LIN {X 157.37, Y 132.33, Z 0.00, A 0, B 0, C 0} C_DIS
LIN {X 157.50, Y 132.59, Z 0.00, A 0, B 0, C 0} C_DIS
LIN {X 157.62, Y 132.87, Z 0.00, A 0, B 0, C 0} C_DIS
LIN {X 157.74, Y 133.14, Z 0.00, A 0, B 0, C 0} C_DIS
LIN {X 157.86, Y 133.42, Z 0.00, A 0, B 0, C 0} C_DIS
LIN {X 157.98, Y 133.69, Z 0.00, A 0, B 0, C 0} C_DIS
LIN {X 158.10, Y 133.97, Z 0.00, A 0, B 0, C 0} C_DIS
LIN {X 158.22, Y 134.24, Z 0.00, A 0, B 0, C 0} C_DIS
LIN {X 158.34, Y 134.51, Z 0.00, A 0, B 0, C 0} C_DIS
LIN {X 158.47, Y 134.78, Z 0.00, A 0, B 0, C 0} C_DIS
LIN {X 158.59, Y 135.05, Z 0.00, A 0, B 0, C 0} C_DIS
LIN {X 158.70, Y 135.33, Z 0.00, A 0, B 0, C 0} C_DIS
LIN {X 158.80, Y 135.62, Z 0.00, A 0, B 0, C 0} C_DIS
LIN {X 158.89, Y 135.92, Z 0.00, A 0, B 0, C 0} C_DIS
LIN {X 158.97, Y 136.22, Z 0.00, A 0, B 0, C 0} C_DIS
LIN {X 159.08, Y 136.51, Z 0.00, A 0, B 0, C 0} C_DIS
LIN {X 159.20, Y 136.78, Z 0.00, A 0, B 0, C 0} C_DIS
LIN {X 159.32, Y 137.05, Z 0.00, A 0, B 0, C 0} C_DIS
LIN {X 159.44, Y 137.32, Z 0.00, A 0, B 0, C 0} C_DIS
LIN {X 159.56, Y 137.60, Z 0.00, A 0, B 0, C 0} C_DIS
LIN {X 159.68, Y 137.87, Z 0.00, A 0, B 0, C 0} C_DIS
LIN {X 159.80, Y 138.14, Z 0.00, A 0, B 0, C 0} C_DIS
LIN {X 159.93, Y 138.41, Z 0.00, A 0, B 0, C 0} C_DIS
LIN {X 160.04, Y 138.69, Z 0.00, A 0, B 0, C 0} C_DIS
LIN {X 160.14, Y 138.98, Z 0.00, A 0, B 0, C 0} C_DIS
LIN {X 160.22, Y 139.29, Z 0.00, A 0, B 0, C 0} C_DIS
LIN {X 160.31, Y 139.58, Z 0.00, A 0, B 0, C 0} C_DIS
LIN {X 160.42, Y 139.86, Z 0.00, A 0, B 0, C 0} C_DIS
LIN {X 160.53, Y 140.14, Z 0.00, A 0, B 0, C 0} C_DIS
LIN {X 160.61, Y 140.45, Z 0.00, A 0, B 0, C 0} C_DIS
LIN {X 160.67, Y 140.76, Z 0.00, A 0, B 0, C 0} C_DIS
LIN {X 160.73, Y 141.08, Z 0.00, A 0, B 0, C 0} C_DIS
LIN {X 160.82, Y 141.38, Z 0.00, A 0, B 0, C 0} C_DIS
LIN {X 160.90, Y 141.68, Z 0.00, A 0, B 0, C 0} C_DIS
LIN {X 160.98, Y 141.99, Z 0.00, A 0, B 0, C 0} C_DIS
LIN {X 161.04, Y 142.30, Z 0.00, A 0, B 0, C 0} C_DIS
LIN {X 161.10, Y 142.61, Z 0.00, A 0, B 0, C 0} C_DIS
LIN {X 161.19, Y 142.91, Z 0.00, A 0, B 0, C 0} C_DIS
LIN {X 161.31, Y 143.19, Z 0.00, A 0, B 0, C 0} C_DIS
LIN {X 161.42, Y 143.47, Z 0.00, A 0, B 0, C 0} C_DIS
LIN {X 161.49, Y 143.78, Z 0.00, A 0, B 0, C 0} C_DIS
LIN {X 161.55, Y 144.09, Z 0.00, A 0, B 0, C 0} C_DIS
LIN {X 161.61, Y 144.40, Z 0.00, A 0, B 0, C 0} C_DIS
LIN {X 161.70, Y 144.71, Z 0.00, A 0, B 0, C 0} C_DIS
LIN {X 161.79, Y 145.00, Z 0.00, A 0, B 0, C 0} C_DIS
LIN {X 161.86, Y 145.31, Z 0.00, A 0, B 0, C 0} C_DIS
LIN {X 161.91, Y 145.63, Z 0.00, A 0, B 0, C 0} C_DIS
LIN {X 161.96, Y 145.95, Z 0.00, A 0, B 0, C 0} C_DIS
LIN {X 162.02, Y 146.27, Z 0.00, A 0, B 0, C 0} C_DIS
LIN {X 162.10, Y 146.57, Z 0.00, A 0, B 0, C 0} C_DIS
LIN {X 162.19, Y 146.87, Z 0.00, A 0, B 0, C 0} C_DIS
LIN {X 162.27, Y 147.17, Z 0.00, A 0, B 0, C 0} C_DIS
LIN {X 162.33, Y 147.49, Z 0.00, A 0, B 0, C 0} C_DIS
LIN {X 162.38, Y 147.81, Z 0.00, A 0, B 0, C 0} C_DIS
LIN {X 162.44, Y 148.12, Z 0.00, A 0, B 0, C 0} C_DIS
LIN {X 162.49, Y 148.44, Z 0.00, A 0, B 0, C 0} C_DIS
LIN {X 162.53, Y 148.76, Z 0.00, A 0, B 0, C 0} C_DIS
LIN {X 162.56, Y 149.08, Z 0.00, A 0, B 0, C 0} C_DIS
LIN {X 162.59, Y 149.41, Z 0.00, A 0, B 0, C 0} C_DIS
LIN {X 162.61, Y 149.74, Z 0.00, A 0, B 0, C 0} C_DIS
LIN {X 162.64, Y 150.06, Z 0.00, A 0, B 0, C 0} C_DIS
LIN {X 162.69, Y 150.38, Z 0.00, A 0, B 0, C 0} C_DIS
LIN {X 162.75, Y 150.70, Z 0.00, A 0, B 0, C 0} C_DIS
LIN {X 162.81, Y 151.01, Z 0.00, A 0, B 0, C 0} C_DIS
LIN {X 162.86, Y 151.33, Z 0.00, A 0, B 0, C 0} C_DIS
LIN {X 162.92, Y 151.65, Z 0.00, A 0, B 0, C 0} C_DIS
LIN {X 162.96, Y 151.97, Z 0.00, A 0, B 0, C 0} C_DIS
LIN {X 163.00, Y 152.29, Z 0.00, A 0, B 0, C 0} C_DIS
LIN {X 163.01, Y 152.61, Z 0.00, A 0, B 0, C 0} C_DIS
LIN {X 163.02, Y 152.94, Z 0.00, A 0, B 0, C 0} C_DIS
LIN {X 163.01, Y 153.27, Z 0.00, A 0, B 0, C 0} C_DIS
LIN {X 163.00, Y 153.60, Z 0.00, A 0, B 0, C 0} C_DIS
LIN {X 163.01, Y 153.93, Z 0.00, A 0, B 0, C 0} C_DIS
LIN {X 163.03, Y 154.25, Z 0.00, A 0, B 0, C 0} C_DIS
LIN {X 163.07, Y 154.58, Z 0.00, A 0, B 0, C 0} C_DIS
LIN {X 163.12, Y 154.89, Z 0.00, A 0, B 0, C 0} C_DIS
LIN {X 163.18, Y 155.21, Z 0.00, A 0, B 0, C 0} C_DIS
LIN {X 163.24, Y 155.53, Z 0.00, A 0, B 0, C 0} C_DIS
LIN {X 163.29, Y 155.85, Z 0.00, A 0, B 0, C 0} C_DIS
LIN {X 163.34, Y 156.17, Z 0.00, A 0, B 0, C 0} C_DIS
LIN {X 163.38, Y 156.49, Z 0.00, A 0, B 0, C 0} C_DIS
LIN {X 163.41, Y 156.81, Z 0.00, A 0, B 0, C 0} C_DIS
LIN {X 163.43, Y 157.13, Z 0.00, A 0, B 0, C 0} C_DIS
LIN {X 163.45, Y 157.46, Z 0.00, A 0, B 0, C 0} C_DIS
LIN {X 163.45, Y 157.79, Z 0.00, A 0, B 0, C 0} C_DIS
LIN {X 163.46, Y 158.11, Z 0.00, A 0, B 0, C 0} C_DIS
LIN {X 163.46, Y 158.44, Z 0.00, A 0, B 0, C 0} C_DIS
LIN {X 163.45, Y 158.77, Z 0.00, A 0, B 0, C 0} C_DIS
LIN {X 163.45, Y 159.10, Z 0.00, A 0, B 0, C 0} C_DIS
LIN {X 163.44, Y 159.43, Z 0.00, A 0, B 0, C 0} C_DIS
LIN {X 163.44, Y 159.75, Z 0.00, A 0, B 0, C 0} C_DIS
LIN {X 163.43, Y 160.08, Z 0.00, A 0, B 0, C 0} C_DIS
LIN {X 163.44, Y 160.41, Z 0.00, A 0, B 0, C 0} C_DIS
LIN {X 163.45, Y 160.74, Z 0.00, A 0, B 0, C 0} C_DIS
LIN {X 163.46, Y 161.07, Z 0.00, A 0, B 0, C 0} C_DIS
LIN {X 163.46, Y 161.40, Z 0.00, A 0, B 0, C 0} C_DIS
LIN {X 163.46, Y 161.72, Z 0.00, A 0, B 0, C 0} C_DIS
LIN {X 163.44, Y 162.05, Z 0.00, A 0, B 0, C 0} C_DIS
LIN {X 163.40, Y 162.37, Z 0.00, A 0, B 0, C 0} C_DIS
LIN {X 163.36, Y 162.69, Z 0.00, A 0, B 0, C 0} C_DIS
LIN {X 163.30, Y 163.01, Z 0.00, A 0, B 0, C 0} C_DIS
LIN {X 163.25, Y 163.33, Z 0.00, A 0, B 0, C 0} C_DIS
LIN {X 163.19, Y 163.64, Z 0.00, A 0, B 0, C 0} C_DIS
LIN {X 163.14, Y 163.96, Z 0.00, A 0, B 0, C 0} C_DIS
LIN {X 163.09, Y 164.28, Z 0.00, A 0, B 0, C 0} C_DIS
LIN {X 163.05, Y 164.60, Z 0.00, A 0, B 0, C 0} C_DIS
LIN {X 163.03, Y 164.93, Z 0.00, A 0, B 0, C 0} C_DIS
LIN {X 163.02, Y 165.25, Z 0.00, A 0, B 0, C 0} C_DIS
LIN {X 163.01, Y 165.58, Z 0.00, A 0, B 0, C 0} C_DIS
LIN {X 163.01, Y 165.91, Z 0.00, A 0, B 0, C 0} C_DIS
LIN {X 163.01, Y 166.24, Z 0.00, A 0, B 0, C 0} C_DIS
LIN {X 163.01, Y 166.56, Z 0.00, A 0, B 0, C 0} C_DIS
LIN {X 163.02, Y 166.89, Z 0.00, A 0, B 0, C 0} C_DIS
LIN {X 163.01, Y 167.22, Z 0.00, A 0, B 0, C 0} C_DIS
LIN {X 163.00, Y 167.55, Z 0.00, A 0, B 0, C 0} C_DIS
LIN {X 162.99, Y 167.87, Z 0.00, A 0, B 0, C 0} C_DIS
LIN {X 162.97, Y 168.20, Z 0.00, A 0, B 0, C 0} C_DIS
LIN {X 162.94, Y 168.52, Z 0.00, A 0, B 0, C 0} C_DIS
LIN {X 162.89, Y 168.84, Z 0.00, A 0, B 0, C 0} C_DIS
LIN {X 162.84, Y 169.16, Z 0.00, A 0, B 0, C 0} C_DIS
LIN {X 162.78, Y 169.47, Z 0.00, A 0, B 0, C 0} C_DIS
LIN {X 162.72, Y 169.79, Z 0.00, A 0, B 0, C 0} C_DIS
LIN {X 162.67, Y 170.11, Z 0.00, A 0, B 0, C 0} C_DIS
LIN {X 162.61, Y 170.43, Z 0.00, A 0, B 0, C 0} C_DIS
LIN {X 162.56, Y 170.74, Z 0.00, A 0, B 0, C 0} C_DIS
LIN {X 162.51, Y 171.06, Z 0.00, A 0, B 0, C 0} C_DIS
LIN {X 162.46, Y 171.38, Z 0.00, A 0, B 0, C 0} C_DIS
LIN {X 162.41, Y 171.70, Z 0.00, A 0, B 0, C 0} C_DIS
LIN {X 162.36, Y 172.02, Z 0.00, A 0, B 0, C 0} C_DIS
LIN {X 162.30, Y 172.33, Z 0.00, A 0, B 0, C 0} C_DIS
LIN {X 162.25, Y 172.65, Z 0.00, A 0, B 0, C 0} C_DIS
LIN {X 162.20, Y 172.97, Z 0.00, A 0, B 0, C 0} C_DIS
LIN {X 162.14, Y 173.29, Z 0.00, A 0, B 0, C 0} C_DIS
LIN {X 162.09, Y 173.61, Z 0.00, A 0, B 0, C 0} C_DIS
LIN {X 162.04, Y 173.92, Z 0.00, A 0, B 0, C 0} C_DIS
LIN {X 161.98, Y 174.24, Z 0.00, A 0, B 0, C 0} C_DIS
LIN {X 161.93, Y 174.56, Z 0.00, A 0, B 0, C 0} C_DIS
LIN {X 161.88, Y 174.88, Z 0.00, A 0, B 0, C 0} C_DIS
LIN {X 161.82, Y 175.19, Z 0.00, A 0, B 0, C 0} C_DIS
LIN {X 161.74, Y 175.50, Z 0.00, A 0, B 0, C 0} C_DIS
LIN {X 161.64, Y 175.79, Z 0.00, A 0, B 0, C 0} C_DIS
LIN {X 161.57, Y 176.10, Z 0.00, A 0, B 0, C 0} C_DIS
LIN {X 161.52, Y 176.42, Z 0.00, A 0, B 0, C 0} C_DIS
LIN {X 161.47, Y 176.74, Z 0.00, A 0, B 0, C 0} C_DIS
LIN {X 161.40, Y 177.05, Z 0.00, A 0, B 0, C 0} C_DIS
LIN {X 161.32, Y 177.35, Z 0.00, A 0, B 0, C 0} C_DIS
LIN {X 161.24, Y 177.66, Z 0.00, A 0, B 0, C 0} C_DIS
LIN {X 161.17, Y 177.96, Z 0.00, A 0, B 0, C 0} C_DIS
LIN {X 161.10, Y 178.27, Z 0.00, A 0, B 0, C 0} C_DIS
LIN {X 161.03, Y 178.58, Z 0.00, A 0, B 0, C 0} C_DIS
LIN {X 160.95, Y 178.89, Z 0.00, A 0, B 0, C 0} C_DIS
LIN {X 160.84, Y 179.17, Z 0.00, A 0, B 0, C 0} C_DIS
LIN {X 160.73, Y 179.45, Z 0.00, A 0, B 0, C 0} C_DIS
LIN {X 160.65, Y 179.75, Z 0.00, A 0, B 0, C 0} C_DIS
LIN {X 160.58, Y 180.06, Z 0.00, A 0, B 0, C 0} C_DIS
LIN {X 160.52, Y 180.37, Z 0.00, A 0, B 0, C 0} C_DIS
LIN {X 160.45, Y 180.68, Z 0.00, A 0, B 0, C 0} C_DIS
LIN {X 160.37, Y 180.99, Z 0.00, A 0, B 0, C 0} C_DIS
LIN {X 160.28, Y 181.29, Z 0.00, A 0, B 0, C 0} C_DIS
LIN {X 160.18, Y 181.58, Z 0.00, A 0, B 0, C 0} C_DIS
LIN {X 160.08, Y 181.87, Z 0.00, A 0, B 0, C 0} C_DIS
LIN {X 159.96, Y 182.14, Z 0.00, A 0, B 0, C 0} C_DIS
LIN {X 159.84, Y 182.42, Z 0.00, A 0, B 0, C 0} C_DIS
LIN {X 159.72, Y 182.69, Z 0.00, A 0, B 0, C 0} C_DIS
LIN {X 159.59, Y 182.96, Z 0.00, A 0, B 0, C 0} C_DIS
LIN {X 159.48, Y 183.23, Z 0.00, A 0, B 0, C 0} C_DIS
LIN {X 159.38, Y 183.53, Z 0.00, A 0, B 0, C 0} C_DIS
LIN {X 159.30, Y 183.83, Z 0.00, A 0, B 0, C 0} C_DIS
LIN {X 159.21, Y 184.13, Z 0.00, A 0, B 0, C 0} C_DIS
LIN {X 159.11, Y 184.41, Z 0.00, A 0, B 0, C 0} C_DIS
LIN {X 159.00, Y 184.70, Z 0.00, A 0, B 0, C 0} C_DIS
LIN {X 158.90, Y 184.99, Z 0.00, A 0, B 0, C 0} C_DIS
LIN {X 158.82, Y 185.29, Z 0.00, A 0, B 0, C 0} C_DIS
LIN {X 158.73, Y 185.59, Z 0.00, A 0, B 0, C 0} C_DIS
LIN {X 158.61, Y 185.87, Z 0.00, A 0, B 0, C 0} C_DIS
LIN {X 158.49, Y 186.13, Z 0.00, A 0, B 0, C 0} C_DIS
LIN {X 158.36, Y 186.41, Z 0.00, A 0, B 0, C 0} C_DIS
LIN {X 158.24, Y 186.67, Z 0.00, A 0, B 0, C 0} C_DIS
LIN {X 158.09, Y 186.91, Z 0.00, A 0, B 0, C 0} C_DIS
LIN {X 157.93, Y 187.14, Z 0.00, A 0, B 0, C 0} C_DIS
LIN {X 157.79, Y 187.38, Z 0.00, A 0, B 0, C 0} C_DIS
LIN {X 157.66, Y 187.65, Z 0.00, A 0, B 0, C 0} C_DIS
LIN {X 157.54, Y 187.92, Z 0.00, A 0, B 0, C 0} C_DIS
LIN {X 157.42, Y 188.20, Z 0.00, A 0, B 0, C 0} C_DIS
LIN {X 157.31, Y 188.48, Z 0.00, A 0, B 0, C 0} C_DIS
LIN {X 157.19, Y 188.75, Z 0.00, A 0, B 0, C 0} C_DIS
LIN {X 157.06, Y 189.02, Z 0.00, A 0, B 0, C 0} C_DIS
LIN {X 156.93, Y 189.28, Z 0.00, A 0, B 0, C 0} C_DIS
LIN {X 156.79, Y 189.53, Z 0.00, A 0, B 0, C 0} C_DIS
LIN {X 156.64, Y 189.76, Z 0.00, A 0, B 0, C 0} C_DIS
LIN {X 156.48, Y 189.98, Z 0.00, A 0, B 0, C 0} C_DIS
LIN {X 156.32, Y 190.21, Z 0.00, A 0, B 0, C 0} C_DIS
LIN {X 156.17, Y 190.45, Z 0.00, A 0, B 0, C 0} C_DIS
LIN {X 156.04, Y 190.70, Z 0.00, A 0, B 0, C 0} C_DIS
LIN {X 155.91, Y 190.96, Z 0.00, A 0, B 0, C 0} C_DIS
LIN {X 155.79, Y 191.23, Z 0.00, A 0, B 0, C 0} C_DIS
LIN {X 155.67, Y 191.51, Z 0.00, A 0, B 0, C 0} C_DIS
LIN {X 155.55, Y 191.79, Z 0.00, A 0, B 0, C 0} C_DIS
LIN {X 155.43, Y 192.06, Z 0.00, A 0, B 0, C 0} C_DIS
LIN {X 155.31, Y 192.33, Z 0.00, A 0, B 0, C 0} C_DIS
LIN {X 155.18, Y 192.59, Z 0.00, A 0, B 0, C 0} C_DIS
LIN {X 155.03, Y 192.83, Z 0.00, A 0, B 0, C 0} C_DIS
LIN {X 154.88, Y 193.07, Z 0.00, A 0, B 0, C 0} C_DIS
LIN {X 154.72, Y 193.29, Z 0.00, A 0, B 0, C 0} C_DIS
LIN {X 154.57, Y 193.52, Z 0.00, A 0, B 0, C 0} C_DIS
LIN {X 154.41, Y 193.75, Z 0.00, A 0, B 0, C 0} C_DIS
LIN {X 154.26, Y 193.98, Z 0.00, A 0, B 0, C 0} C_DIS
LIN {X 154.11, Y 194.22, Z 0.00, A 0, B 0, C 0} C_DIS
LIN {X 153.96, Y 194.46, Z 0.00, A 0, B 0, C 0} C_DIS
LIN {X 153.80, Y 194.69, Z 0.00, A 0, B 0, C 0} C_DIS
LIN {X 153.64, Y 194.90, Z 0.00, A 0, B 0, C 0} C_DIS
LIN {X 153.46, Y 195.09, Z 0.00, A 0, B 0, C 0} C_DIS
LIN {X 153.28, Y 195.27, Z 0.00, A 0, B 0, C 0} C_DIS
LIN {X 153.09, Y 195.44, Z 0.00, A 0, B 0, C 0} C_DIS
LIN {X 152.91, Y 195.62, Z 0.00, A 0, B 0, C 0} C_DIS
LIN {X 152.73, Y 195.81, Z 0.00, A 0, B 0, C 0} C_DIS
LIN {X 152.56, Y 196.00, Z 0.00, A 0, B 0, C 0} C_DIS
LIN {X 152.38, Y 196.20, Z 0.00, A 0, B 0, C 0} C_DIS
LIN {X 152.22, Y 196.41, Z 0.00, A 0, B 0, C 0} C_DIS
LIN {X 152.06, Y 196.63, Z 0.00, A 0, B 0, C 0} C_DIS
LIN {X 151.91, Y 196.86, Z 0.00, A 0, B 0, C 0} C_DIS
LIN {X 151.76, Y 197.10, Z 0.00, A 0, B 0, C 0} C_DIS
LIN {X 151.61, Y 197.34, Z 0.00, A 0, B 0, C 0} C_DIS
LIN {X 151.46, Y 197.58, Z 0.00, A 0, B 0, C 0} C_DIS
LIN {X 151.30, Y 197.81, Z 0.00, A 0, B 0, C 0} C_DIS
LIN {X 151.14, Y 198.03, Z 0.00, A 0, B 0, C 0} C_DIS
LIN {X 150.97, Y 198.23, Z 0.00, A 0, B 0, C 0} C_DIS
LIN {X 150.80, Y 198.42, Z 0.00, A 0, B 0, C 0} C_DIS
LIN {X 150.62, Y 198.60, Z 0.00, A 0, B 0, C 0} C_DIS
LIN {X 150.43, Y 198.78, Z 0.00, A 0, B 0, C 0} C_DIS
LIN {X 150.25, Y 198.95, Z 0.00, A 0, B 0, C 0} C_DIS
LIN {X 150.07, Y 199.14, Z 0.00, A 0, B 0, C 0} C_DIS
LIN {X 149.89, Y 199.33, Z 0.00, A 0, B 0, C 0} C_DIS
LIN {X 149.72, Y 199.53, Z 0.00, A 0, B 0, C 0} C_DIS
LIN {X 149.56, Y 199.75, Z 0.00, A 0, B 0, C 0} C_DIS
LIN {X 149.41, Y 199.98, Z 0.00, A 0, B 0, C 0} C_DIS
LIN {X 149.24, Y 200.20, Z 0.00, A 0, B 0, C 0} C_DIS
LIN {X 149.07, Y 200.38, Z 0.00, A 0, B 0, C 0} C_DIS
LIN {X 148.88, Y 200.56, Z 0.00, A 0, B 0, C 0} C_DIS
LIN {X 148.70, Y 200.74, Z 0.00, A 0, B 0, C 0} C_DIS
LIN {X 148.52, Y 200.92, Z 0.00, A 0, B 0, C 0} C_DIS
LIN {X 148.34, Y 201.10, Z 0.00, A 0, B 0, C 0} C_DIS
LIN {X 148.16, Y 201.28, Z 0.00, A 0, B 0, C 0} C_DIS
LIN {X 147.98, Y 201.46, Z 0.00, A 0, B 0, C 0} C_DIS
LIN {X 147.80, Y 201.65, Z 0.00, A 0, B 0, C 0} C_DIS
LIN {X 147.62, Y 201.83, Z 0.00, A 0, B 0, C 0} C_DIS
LIN {X 147.43, Y 202.01, Z 0.00, A 0, B 0, C 0} C_DIS
LIN {X 147.25, Y 202.19, Z 0.00, A 0, B 0, C 0} C_DIS
LIN {X 147.07, Y 202.37, Z 0.00, A 0, B 0, C 0} C_DIS
LIN {X 146.89, Y 202.55, Z 0.00, A 0, B 0, C 0} C_DIS
LIN {X 146.71, Y 202.73, Z 0.00, A 0, B 0, C 0} C_DIS
LIN {X 146.53, Y 202.92, Z 0.00, A 0, B 0, C 0} C_DIS
LIN {X 146.35, Y 203.10, Z 0.00, A 0, B 0, C 0} C_DIS
LIN {X 146.16, Y 203.28, Z 0.00, A 0, B 0, C 0} C_DIS
LIN {X 145.98, Y 203.46, Z 0.00, A 0, B 0, C 0} C_DIS
LIN {X 145.81, Y 203.65, Z 0.00, A 0, B 0, C 0} C_DIS
LIN {X 145.63, Y 203.83, Z 0.00, A 0, B 0, C 0} C_DIS
LIN {X 145.45, Y 204.02, Z 0.00, A 0, B 0, C 0} C_DIS
LIN {X 145.28, Y 204.23, Z 0.00, A 0, B 0, C 0} C_DIS
LIN {X 145.12, Y 204.45, Z 0.00, A 0, B 0, C 0} C_DIS
LIN {X 144.97, Y 204.69, Z 0.00, A 0, B 0, C 0} C_DIS
LIN {X 144.83, Y 204.94, Z 0.00, A 0, B 0, C 0} C_DIS
LIN {X 144.70, Y 205.19, Z 0.00, A 0, B 0, C 0} C_DIS
LIN {X 144.57, Y 205.45, Z 0.00, A 0, B 0, C 0} C_DIS
LIN {X 144.44, Y 205.72, Z 0.00, A 0, B 0, C 0} C_DIS
LIN {X 144.32, Y 206.00, Z 0.00, A 0, B 0, C 0} C_DIS
LIN {X 144.22, Y 206.29, Z 0.00, A 0, B 0, C 0} C_DIS
LIN {X 144.13, Y 206.59, Z 0.00, A 0, B 0, C 0} C_DIS
LIN {X 144.06, Y 206.89, Z 0.00, A 0, B 0, C 0} C_DIS
LIN {X 144.00, Y 207.21, Z 0.00, A 0, B 0, C 0} C_DIS
LIN {X 143.95, Y 207.53, Z 0.00, A 0, B 0, C 0} C_DIS
LIN {X 143.92, Y 207.85, Z 0.00, A 0, B 0, C 0} C_DIS
LIN {X 143.89, Y 208.18, Z 0.00, A 0, B 0, C 0} C_DIS
LIN {X 143.87, Y 208.50, Z 0.00, A 0, B 0, C 0} C_DIS
LIN {X 143.87, Y 208.83, Z 0.00, A 0, B 0, C 0} C_DIS
LIN {X 143.87, Y 209.16, Z 0.00, A 0, B 0, C 0} C_DIS
LIN {X 143.87, Y 209.49, Z 0.00, A 0, B 0, C 0} C_DIS
LIN {X 143.88, Y 209.82, Z 0.00, A 0, B 0, C 0} C_DIS
LIN {X 143.88, Y 210.14, Z 0.00, A 0, B 0, C 0} C_DIS
LIN {X 143.87, Y 210.47, Z 0.00, A 0, B 0, C 0} C_DIS
LIN {X 143.84, Y 210.79, Z 0.00, A 0, B 0, C 0} C_DIS
LIN {X 143.80, Y 211.12, Z 0.00, A 0, B 0, C 0} C_DIS
LIN {X 143.75, Y 211.43, Z 0.00, A 0, B 0, C 0} C_DIS
LIN {X 143.70, Y 211.75, Z 0.00, A 0, B 0, C 0} C_DIS
LIN {X 143.64, Y 212.07, Z 0.00, A 0, B 0, C 0} C_DIS
LIN {X 143.58, Y 212.38, Z 0.00, A 0, B 0, C 0} C_DIS
LIN {X 143.53, Y 212.70, Z 0.00, A 0, B 0, C 0} C_DIS
LIN {X 143.49, Y 213.02, Z 0.00, A 0, B 0, C 0} C_DIS
LIN {X 143.46, Y 213.35, Z 0.00, A 0, B 0, C 0} C_DIS
LIN {X 143.44, Y 213.67, Z 0.00, A 0, B 0, C 0} C_DIS
LIN {X 143.43, Y 214.00, Z 0.00, A 0, B 0, C 0} C_DIS
LIN {X 143.43, Y 214.33, Z 0.00, A 0, B 0, C 0} C_DIS
LIN {X 143.44, Y 214.66, Z 0.00, A 0, B 0, C 0} C_DIS
LIN {X 143.44, Y 214.99, Z 0.00, A 0, B 0, C 0} C_DIS
LIN {X 143.45, Y 215.31, Z 0.00, A 0, B 0, C 0} C_DIS
LIN {X 143.44, Y 215.64, Z 0.00, A 0, B 0, C 0} C_DIS
LIN {X 143.41, Y 215.97, Z 0.00, A 0, B 0, C 0} C_DIS
LIN {X 143.38, Y 216.29, Z 0.00, A 0, B 0, C 0} C_DIS
LIN {X 143.33, Y 216.61, Z 0.00, A 0, B 0, C 0} C_DIS
LIN {X 143.27, Y 216.92, Z 0.00, A 0, B 0, C 0} C_DIS
LIN {X 143.22, Y 217.24, Z 0.00, A 0, B 0, C 0} C_DIS
LIN {X 143.16, Y 217.56, Z 0.00, A 0, B 0, C 0} C_DIS
LIN {X 143.11, Y 217.88, Z 0.00, A 0, B 0, C 0} C_DIS
LIN {X 143.06, Y 218.20, Z 0.00, A 0, B 0, C 0} C_DIS
LIN {X 143.03, Y 218.52, Z 0.00, A 0, B 0, C 0} C_DIS
LIN {X 143.00, Y 218.84, Z 0.00, A 0, B 0, C 0} C_DIS
LIN {X 143.00, Y 219.17, Z 0.00, A 0, B 0, C 0} C_DIS
LIN {X 143.00, Y 219.50, Z 0.00, A 0, B 0, C 0} C_DIS
LIN {X 143.00, Y 219.83, Z 0.00, A 0, B 0, C 0} C_DIS
LIN {X 143.01, Y 220.16, Z 0.00, A 0, B 0, C 0} C_DIS
LIN {X 143.01, Y 220.48, Z 0.00, A 0, B 0, C 0} C_DIS
LIN {X 143.00, Y 220.81, Z 0.00, A 0, B 0, C 0} C_DIS
LIN {X 142.98, Y 221.14, Z 0.00, A 0, B 0, C 0} C_DIS
LIN {X 142.95, Y 221.46, Z 0.00, A 0, B 0, C 0} C_DIS
LIN {X 142.91, Y 221.78, Z 0.00, A 0, B 0, C 0} C_DIS
LIN {X 142.85, Y 222.10, Z 0.00, A 0, B 0, C 0} C_DIS
LIN {X 142.79, Y 222.41, Z 0.00, A 0, B 0, C 0} C_DIS
LIN {X 142.74, Y 222.73, Z 0.00, A 0, B 0, C 0} C_DIS
LIN {X 142.68, Y 223.05, Z 0.00, A 0, B 0, C 0} C_DIS
LIN {X 142.64, Y 223.37, Z 0.00, A 0, B 0, C 0} C_DIS
LIN {X 142.60, Y 223.69, Z 0.00, A 0, B 0, C 0} C_DIS
LIN {X 142.57, Y 224.02, Z 0.00, A 0, B 0, C 0} C_DIS
LIN {X 142.56, Y 224.34, Z 0.00, A 0, B 0, C 0} C_DIS
LIN {X 142.56, Y 224.67, Z 0.00, A 0, B 0, C 0} C_DIS
LIN {X 142.57, Y 225.00, Z 0.00, A 0, B 0, C 0} C_DIS
LIN {X 142.57, Y 225.33, Z 0.00, A 0, B 0, C 0} C_DIS
LIN {X 142.58, Y 225.66, Z 0.00, A 0, B 0, C 0} C_DIS
LIN {X 142.57, Y 225.98, Z 0.00, A 0, B 0, C 0} C_DIS
LIN {X 142.55, Y 226.31, Z 0.00, A 0, B 0, C 0} C_DIS
LIN {X 142.53, Y 226.63, Z 0.00, A 0, B 0, C 0} C_DIS
LIN {X 142.48, Y 226.95, Z 0.00, A 0, B 0, C 0} C_DIS
LIN {X 142.43, Y 227.27, Z 0.00, A 0, B 0, C 0} C_DIS
LIN {X 142.37, Y 227.59, Z 0.00, A 0, B 0, C 0} C_DIS
LIN {X 142.31, Y 227.90, Z 0.00, A 0, B 0, C 0} C_DIS
LIN {X 142.26, Y 228.22, Z 0.00, A 0, B 0, C 0} C_DIS
LIN {X 142.21, Y 228.54, Z 0.00, A 0, B 0, C 0} C_DIS
LIN {X 142.17, Y 228.86, Z 0.00, A 0, B 0, C 0} C_DIS
LIN {X 142.14, Y 229.19, Z 0.00, A 0, B 0, C 0} C_DIS
LIN {X 142.13, Y 229.51, Z 0.00, A 0, B 0, C 0} C_DIS
LIN {X 142.13, Y 229.84, Z 0.00, A 0, B 0, C 0} C_DIS
LIN {X 142.13, Y 230.17, Z 0.00, A 0, B 0, C 0} C_DIS
LIN {X 142.14, Y 230.50, Z 0.00, A 0, B 0, C 0} C_DIS
LIN {X 142.14, Y 230.83, Z 0.00, A 0, B 0, C 0} C_DIS
LIN {X 142.14, Y 231.15, Z 0.00, A 0, B 0, C 0} C_DIS
LIN {X 142.12, Y 231.48, Z 0.00, A 0, B 0, C 0} C_DIS
LIN {X 142.10, Y 231.81, Z 0.00, A 0, B 0, C 0} C_DIS
LIN {X 142.06, Y 232.13, Z 0.00, A 0, B 0, C 0} C_DIS
LIN {X 142.01, Y 232.44, Z 0.00, A 0, B 0, C 0} C_DIS
LIN {X 141.95, Y 232.76, Z 0.00, A 0, B 0, C 0} C_DIS
LIN {X 141.89, Y 233.08, Z 0.00, A 0, B 0, C 0} C_DIS
LIN {X 141.84, Y 233.40, Z 0.00, A 0, B 0, C 0} C_DIS
LIN {X 141.79, Y 233.72, Z 0.00, A 0, B 0, C 0} C_DIS
LIN {X 141.74, Y 234.04, Z 0.00, A 0, B 0, C 0} C_DIS
LIN {X 141.71, Y 234.36, Z 0.00, A 0, B 0, C 0} C_DIS
LIN {X 141.70, Y 234.68, Z 0.00, A 0, B 0, C 0} C_DIS
LIN {X 141.69, Y 235.01, Z 0.00, A 0, B 0, C 0} C_DIS
LIN {X 141.70, Y 235.34, Z 0.00, A 0, B 0, C 0} C_DIS
LIN {X 141.70, Y 235.67, Z 0.00, A 0, B 0, C 0} C_DIS
LIN {X 141.71, Y 236.00, Z 0.00, A 0, B 0, C 0} C_DIS
LIN {X 141.70, Y 236.33, Z 0.00, A 0, B 0, C 0} C_DIS
LIN {X 141.69, Y 236.65, Z 0.00, A 0, B 0, C 0} C_DIS
LIN {X 141.67, Y 236.98, Z 0.00, A 0, B 0, C 0} C_DIS
LIN {X 141.63, Y 237.30, Z 0.00, A 0, B 0, C 0} C_DIS
LIN {X 141.59, Y 237.62, Z 0.00, A 0, B 0, C 0} C_DIS
LIN {X 141.53, Y 237.93, Z 0.00, A 0, B 0, C 0} C_DIS
LIN {X 141.47, Y 238.25, Z 0.00, A 0, B 0, C 0} C_DIS
LIN {X 141.41, Y 238.57, Z 0.00, A 0, B 0, C 0} C_DIS
LIN {X 141.36, Y 238.89, Z 0.00, A 0, B 0, C 0} C_DIS
LIN {X 141.31, Y 239.21, Z 0.00, A 0, B 0, C 0} C_DIS
LIN {X 141.29, Y 239.53, Z 0.00, A 0, B 0, C 0} C_DIS
LIN {X 141.27, Y 239.86, Z 0.00, A 0, B 0, C 0} C_DIS
LIN {X 141.27, Y 240.18, Z 0.00, A 0, B 0, C 0} C_DIS
LIN {X 141.26, Y 240.51, Z 0.00, A 0, B 0, C 0} C_DIS
LIN {X 141.26, Y 240.84, Z 0.00, A 0, B 0, C 0} C_DIS
LIN {X 141.25, Y 241.17, Z 0.00, A 0, B 0, C 0} C_DIS
LIN {X 141.26, Y 241.50, Z 0.00, A 0, B 0, C 0} C_DIS
LIN {X 141.27, Y 241.82, Z 0.00, A 0, B 0, C 0} C_DIS
LIN {X 141.30, Y 242.14, Z 0.00, A 0, B 0, C 0} C_DIS
LIN {X 141.34, Y 242.47, Z 0.00, A 0, B 0, C 0} C_DIS
LIN {X 141.38, Y 242.79, Z 0.00, A 0, B 0, C 0} C_DIS
LIN {X 141.43, Y 243.11, Z 0.00, A 0, B 0, C 0} C_DIS
LIN {X 141.49, Y 243.43, Z 0.00, A 0, B 0, C 0} C_DIS
LIN {X 141.58, Y 243.73, Z 0.00, A 0, B 0, C 0} C_DIS
LIN {X 141.70, Y 243.99, Z 0.00, A 0, B 0, C 0} C_DIS
LIN {X 141.85, Y 244.22, Z 0.00, A 0, B 0, C 0} C_DIS
LIN {X 142.01, Y 244.46, Z 0.00, A 0, B 0, C 0} C_DIS
LIN {X 142.16, Y 244.69, Z 0.00, A 0, B 0, C 0} C_DIS
LIN {X 142.33, Y 244.90, Z 0.00, A 0, B 0, C 0} C_DIS
LIN {X 142.52, Y 245.04, Z 0.00, A 0, B 0, C 0} C_DIS
LIN {X 142.72, Y 245.16, Z 0.00, A 0, B 0, C 0} C_DIS
LIN {X 142.92, Y 245.30, Z 0.00, A 0, B 0, C 0} C_DIS
LIN {X 143.10, Y 245.47, Z 0.00, A 0, B 0, C 0} C_DIS
LIN {X 143.29, Y 245.63, Z 0.00, A 0, B 0, C 0} C_DIS
LIN {X 143.50, Y 245.74, Z 0.00, A 0, B 0, C 0} C_DIS
LIN {X 143.70, Y 245.84, Z 0.00, A 0, B 0, C 0} C_DIS
LIN {X 143.91, Y 245.93, Z 0.00, A 0, B 0, C 0} C_DIS
LIN {X 144.13, Y 245.99, Z 0.00, A 0, B 0, C 0} C_DIS
LIN {X 144.34, Y 246.04, Z 0.00, A 0, B 0, C 0} C_DIS
LIN {X 144.56, Y 246.08, Z 0.00, A 0, B 0, C 0} C_DIS
LIN {X 144.78, Y 246.09, Z 0.00, A 0, B 0, C 0} C_DIS
LIN {X 144.99, Y 246.09, Z 0.00, A 0, B 0, C 0} C_DIS
LIN {X 145.21, Y 246.09, Z 0.00, A 0, B 0, C 0} C_DIS
LIN {X 145.43, Y 246.08, Z 0.00, A 0, B 0, C 0} C_DIS
LIN {X 145.65, Y 246.08, Z 0.00, A 0, B 0, C 0} C_DIS
LIN {X 145.86, Y 246.08, Z 0.00, A 0, B 0, C 0} C_DIS
LIN {X 146.08, Y 246.11, Z 0.00, A 0, B 0, C 0} C_DIS
LIN {X 146.29, Y 246.15, Z 0.00, A 0, B 0, C 0} C_DIS
LIN {X 146.51, Y 246.22, Z 0.00, A 0, B 0, C 0} C_DIS
LIN {X 146.72, Y 246.30, Z 0.00, A 0, B 0, C 0} C_DIS
LIN {X 146.93, Y 246.39, Z 0.00, A 0, B 0, C 0} C_DIS
LIN {X 147.14, Y 246.48, Z 0.00, A 0, B 0, C 0} C_DIS
LIN {X 147.35, Y 246.56, Z 0.00, A 0, B 0, C 0} C_DIS
LIN {X 147.56, Y 246.63, Z 0.00, A 0, B 0, C 0} C_DIS
LIN {X 147.77, Y 246.68, Z 0.00, A 0, B 0, C 0} C_DIS
LIN {X 147.99, Y 246.72, Z 0.00, A 0, B 0, C 0} C_DIS
LIN {X 148.21, Y 246.74, Z 0.00, A 0, B 0, C 0} C_DIS
LIN {X 148.42, Y 246.75, Z 0.00, A 0, B 0, C 0} C_DIS
LIN {X 148.64, Y 246.76, Z 0.00, A 0, B 0, C 0} C_DIS
LIN {X 148.86, Y 246.79, Z 0.00, A 0, B 0, C 0} C_DIS
LIN {X 149.07, Y 246.85, Z 0.00, A 0, B 0, C 0} C_DIS
LIN {X 149.28, Y 246.93, Z 0.00, A 0, B 0, C 0} C_DIS
LIN {X 149.49, Y 247.02, Z 0.00, A 0, B 0, C 0} C_DIS
LIN {X 149.70, Y 247.11, Z 0.00, A 0, B 0, C 0} C_DIS
LIN {X 149.91, Y 247.20, Z 0.00, A 0, B 0, C 0} C_DIS
LIN {X 150.12, Y 247.28, Z 0.00, A 0, B 0, C 0} C_DIS
LIN {X 150.33, Y 247.35, Z 0.00, A 0, B 0, C 0} C_DIS
LIN {X 150.54, Y 247.43, Z 0.00, A 0, B 0, C 0} C_DIS
LIN {X 150.76, Y 247.49, Z 0.00, A 0, B 0, C 0} C_DIS
LIN {X 150.97, Y 247.57, Z 0.00, A 0, B 0, C 0} C_DIS
LIN {X 151.18, Y 247.65, Z 0.00, A 0, B 0, C 0} C_DIS
LIN {X 151.39, Y 247.73, Z 0.00, A 0, B 0, C 0} C_DIS
LIN {X 151.60, Y 247.83, Z 0.00, A 0, B 0, C 0} C_DIS
LIN {X 151.80, Y 247.95, Z 0.00, A 0, B 0, C 0} C_DIS
LIN {X 152.00, Y 248.07, Z 0.00, A 0, B 0, C 0} C_DIS
LIN {X 152.20, Y 248.19, Z 0.00, A 0, B 0, C 0} C_DIS
LIN {X 152.41, Y 248.28, Z 0.00, A 0, B 0, C 0} C_DIS
LIN {X 152.62, Y 248.36, Z 0.00, A 0, B 0, C 0} C_DIS
LIN {X 152.83, Y 248.45, Z 0.00, A 0, B 0, C 0} C_DIS
LIN {X 153.04, Y 248.55, Z 0.00, A 0, B 0, C 0} C_DIS
LIN {X 153.24, Y 248.68, Z 0.00, A 0, B 0, C 0} C_DIS
LIN {X 153.44, Y 248.81, Z 0.00, A 0, B 0, C 0} C_DIS
LIN {X 153.64, Y 248.91, Z 0.00, A 0, B 0, C 0} C_DIS
LIN {X 153.85, Y 249.00, Z 0.00, A 0, B 0, C 0} C_DIS
LIN {X 154.06, Y 249.10, Z 0.00, A 0, B 0, C 0} C_DIS
LIN {X 154.25, Y 249.25, Z 0.00, A 0, B 0, C 0} C_DIS
LIN {X 154.43, Y 249.43, Z 0.00, A 0, B 0, C 0} C_DIS
LIN {X 154.63, Y 249.58, Z 0.00, A 0, B 0, C 0} C_DIS
LIN {X 154.83, Y 249.70, Z 0.00, A 0, B 0, C 0} C_DIS
LIN {X 155.03, Y 249.83, Z 0.00, A 0, B 0, C 0} C_DIS
LIN {X 155.22, Y 249.99, Z 0.00, A 0, B 0, C 0} C_DIS
LIN {X 155.40, Y 250.17, Z 0.00, A 0, B 0, C 0} C_DIS
LIN {X 155.58, Y 250.36, Z 0.00, A 0, B 0, C 0} C_DIS
LIN {X 155.75, Y 250.55, Z 0.00, A 0, B 0, C 0} C_DIS
LIN {X 155.94, Y 250.73, Z 0.00, A 0, B 0, C 0} C_DIS
LIN {X 156.12, Y 250.91, Z 0.00, A 0, B 0, C 0} C_DIS
LIN {X 156.30, Y 251.09, Z 0.00, A 0, B 0, C 0} C_DIS
LIN {X 156.49, Y 251.26, Z 0.00, A 0, B 0, C 0} C_DIS
LIN {X 156.67, Y 251.44, Z 0.00, A 0, B 0, C 0} C_DIS
LIN {X 156.84, Y 251.63, Z 0.00, A 0, B 0, C 0} C_DIS
LIN {X 157.02, Y 251.82, Z 0.00, A 0, B 0, C 0} C_DIS
LIN {X 157.19, Y 252.02, Z 0.00, A 0, B 0, C 0} C_DIS
LIN {X 157.35, Y 252.24, Z 0.00, A 0, B 0, C 0} C_DIS
LIN {X 157.51, Y 252.46, Z 0.00, A 0, B 0, C 0} C_DIS
LIN {X 157.67, Y 252.69, Z 0.00, A 0, B 0, C 0} C_DIS
LIN {X 157.82, Y 252.93, Z 0.00, A 0, B 0, C 0} C_DIS
LIN {X 157.97, Y 253.17, Z 0.00, A 0, B 0, C 0} C_DIS
LIN {X 158.12, Y 253.40, Z 0.00, A 0, B 0, C 0} C_DIS
LIN {X 158.27, Y 253.63, Z 0.00, A 0, B 0, C 0} C_DIS
LIN {X 158.43, Y 253.87, Z 0.00, A 0, B 0, C 0} C_DIS
LIN {X 158.58, Y 254.10, Z 0.00, A 0, B 0, C 0} C_DIS
LIN {X 158.73, Y 254.33, Z 0.00, A 0, B 0, C 0} C_DIS
LIN {X 158.89, Y 254.56, Z 0.00, A 0, B 0, C 0} C_DIS
LIN {X 159.05, Y 254.79, Z 0.00, A 0, B 0, C 0} C_DIS
LIN {X 159.20, Y 255.02, Z 0.00, A 0, B 0, C 0} C_DIS
LIN {X 159.36, Y 255.25, Z 0.00, A 0, B 0, C 0} C_DIS
LIN {X 159.51, Y 255.48, Z 0.00, A 0, B 0, C 0} C_DIS
LIN {X 159.66, Y 255.71, Z 0.00, A 0, B 0, C 0} C_DIS
LIN {X 159.81, Y 255.95, Z 0.00, A 0, B 0, C 0} C_DIS
LIN {X 159.95, Y 256.20, Z 0.00, A 0, B 0, C 0} C_DIS
LIN {X 160.09, Y 256.45, Z 0.00, A 0, B 0, C 0} C_DIS
LIN {X 160.22, Y 256.71, Z 0.00, A 0, B 0, C 0} C_DIS
LIN {X 160.34, Y 256.98, Z 0.00, A 0, B 0, C 0} C_DIS
LIN {X 160.46, Y 257.26, Z 0.00, A 0, B 0, C 0} C_DIS
LIN {X 160.55, Y 257.56, Z 0.00, A 0, B 0, C 0} C_DIS
LIN {X 160.62, Y 257.86, Z 0.00, A 0, B 0, C 0} C_DIS
LIN {X 160.68, Y 258.18, Z 0.00, A 0, B 0, C 0} C_DIS
LIN {X 160.72, Y 258.50, Z 0.00, A 0, B 0, C 0} C_DIS
LIN {X 160.73, Y 258.83, Z 0.00, A 0, B 0, C 0} C_DIS
LIN {X 160.73, Y 258.83, Z 10.00, A 0, B 0, C 0}

